C05483=1193.116,-1.564,-43.969,-179.862,5.690,148.965
C05484=1193.121,-1.815,-43.955,-179.864,5.690,148.966
C05485=1193.126,-2.064,-43.941,-179.867,5.690,148.966
C05486=1193.131,-2.313,-43.928,-179.870,5.689,148.967
C05487=1193.136,-2.563,-43.914,-179.872,5.688,148.967
C05488=1193.141,-2.813,-43.900,-179.874,5.688,148.968
C05489=1193.146,-3.062,-43.886,-179.877,5.687,148.969
C05490=1193.151,-3.312,-43.873,-179.880,5.687,148.969
C05491=1193.156,-3.561,-43.859,-179.882,5.686,148.970
C05492=1193.161,-3.811,-43.845,-179.884,5.686,148.971
C05493=1193.166,-4.061,-43.832,-179.887,5.686,148.971
C05494=1193.172,-4.310,-43.818,-179.889,5.685,148.972
C05495=1193.177,-4.560,-43.804,-179.892,5.685,148.973
C05496=1193.182,-4.809,-43.791,-179.895,5.684,148.973
C05497=1193.187,-5.059,-43.777,-179.897,5.683,148.974
C05498=1193.192,-5.309,-43.763,-179.899,5.683,148.974
C05499=1193.197,-5.558,-43.750,-179.902,5.682,148.975
C05500=1193.202,-5.808,-43.736,-179.905,5.682,148.976
C05501=1193.207,-6.057,-43.722,-179.906,5.682,148.976
C05502=1193.212,-6.307,-43.709,-179.909,5.681,148.977
C05503=1193.218,-6.556,-43.695,-179.912,5.681,148.978
C05504=1193.222,-6.806,-43.682,-179.914,5.681,148.978
C05505=1193.227,-7.056,-43.668,-179.917,5.680,148.979
C05506=1193.233,-7.305,-43.655,-179.919,5.679,148.980
C05507=1193.237,-7.555,-43.641,-179.922,5.679,148.980
C05508=1193.243,-7.804,-43.628,-179.924,5.678,148.981
C05509=1193.248,-8.054,-43.614,-179.926,5.679,148.982
C05510=1193.253,-8.303,-43.601,-179.929,5.678,148.982
C05511=1193.258,-8.553,-43.587,-179.931,5.677,148.983
C05512=1193.263,-8.802,-43.574,-179.934,5.677,148.983
C05513=1193.268,-9.052,-43.560,-179.937,5.676,148.984
C05514=1193.273,-9.301,-43.547,-179.939,5.676,148.985
C05515=1193.278,-9.551,-43.533,-179.941,5.675,148.985
C05516=1193.284,-9.801,-43.520,-179.944,5.674,148.986
C05517=1193.289,-10.051,-43.507,-179.946,5.675,148.987
C05518=1193.294,-10.300,-43.493,-179.949,5.674,148.987
C05519=1193.299,-10.550,-43.480,-179.951,5.674,148.988
C05520=1193.304,-10.799,-43.466,-179.954,5.673,148.989
C05521=1193.309,-11.049,-43.453,-179.956,5.673,148.989
C05522=1193.315,-11.298,-43.440,-179.959,5.672,148.990
C05523=1193.319,-11.548,-43.426,-179.962,5.672,148.991
C05524=1193.325,-11.797,-43.413,-179.964,5.672,148.991
C05525=1193.329,-12.048,-43.400,-179.966,5.671,148.992
C05526=1193.335,-12.297,-43.386,-179.968,5.671,148.992
C05527=1193.339,-12.547,-43.373,-179.971,5.670,148.993
C05528=1193.345,-12.796,-43.359,-179.974,5.670,148.994
C05529=1193.349,-13.046,-43.346,-179.976,5.669,148.994
C05530=1193.355,-13.295,-43.333,-179.979,5.668,148.995
C05531=1193.360,-13.545,-43.320,-179.981,5.669,148.996
C05532=1193.365,-13.794,-43.306,-179.983,5.668,148.996
C05533=1193.370,-14.044,-43.293,-179.986,5.668,148.997
C05534=1193.376,-14.294,-43.280,-179.988,5.667,148.998
C05535=1193.380,-14.543,-43.267,-179.991,5.666,148.998
C05536=1193.386,-14.793,-43.253,-179.993,5.666,148.999
C05537=1193.391,-15.042,-43.241,-179.996,5.665,149.000
C05538=1193.395,-15.292,-43.228,-179.998,5.666,149.000
C05539=1193.401,-15.541,-43.214,180.000,5.665,149.001
C05540=1193.405,-15.791,-43.201,179.997,5.664,149.002
C05541=1193.411,-16.041,-43.188,179.994,5.664,149.002
C05542=1193.416,-16.290,-43.175,179.992,5.664,149.003
C05543=1193.421,-16.540,-43.161,179.989,5.663,149.004
C05544=1193.426,-16.789,-43.148,179.987,5.663,149.004
C05545=1193.431,-17.039,-43.135,179.985,5.663,149.005
C05546=1193.437,-17.289,-43.122,179.982,5.662,149.005
C05547=1193.442,-17.538,-43.109,179.979,5.662,149.006
C05548=1193.447,-17.788,-43.096,179.977,5.661,149.007
C05549=1193.452,-18.037,-43.083,179.975,5.660,149.007
C05550=1193.457,-18.287,-43.070,179.973,5.661,149.008
C05551=1193.462,-18.537,-43.056,179.970,5.660,149.009
C05552=1193.468,-18.786,-43.044,179.967,5.660,149.009
C05553=1193.472,-19.036,-43.031,179.965,5.659,149.010
C05554=1193.478,-19.286,-43.018,179.962,5.658,149.011
C05555=1193.483,-19.535,-43.005,179.960,5.658,149.011
C05556=1193.487,-19.785,-42.991,179.958,5.658,149.012
C05557=1193.493,-20.034,-42.978,179.955,5.658,149.013
C05558=1193.498,-20.284,-42.965,179.953,5.657,149.013
C05559=1193.503,-20.534,-42.953,179.950,5.656,149.014
C05560=1193.509,-20.783,-42.939,179.947,5.656,149.014
C05561=1193.513,-21.033,-42.926,179.945,5.656,149.015
C05562=1193.518,-21.282,-42.914,179.943,5.656,149.016
C05563=1193.524,-21.532,-42.901,179.941,5.655,149.016
C05564=1193.529,-21.782,-42.888,179.938,5.655,149.017
C05565=1193.534,-22.031,-42.875,179.935,5.654,149.018
C05566=1193.539,-22.281,-42.862,179.933,5.654,149.018
C05567=1193.544,-22.531,-42.849,179.931,5.654,149.019
C05568=1193.549,-22.780,-42.836,179.928,5.653,149.020
C05569=1193.555,-23.050,-42.822,179.926,5.653,149.020
C05570=1193.561,-23.319,-42.809,179.923,5.652,149.021
C05571=1193.566,-23.590,-42.794,179.920,5.652,149.022
C05572=1193.571,-23.859,-42.780,179.918,5.651,149.022
C05573=1193.576,-24.108,-42.767,179.915,5.651,149.023
C05574=1193.582,-24.358,-42.756,179.912,5.650,149.024
C05575=1193.588,-24.608,-42.742,179.910,5.651,149.024
C05576=1193.592,-24.858,-42.729,179.908,5.650,149.025
C05577=1193.597,-25.107,-42.717,179.905,5.649,149.026
C05578=1193.602,-25.356,-42.704,179.903,5.649,149.026
C05579=1193.608,-25.607,-42.691,179.900,5.648,149.027
C05580=1193.613,-25.856,-42.678,179.898,5.649,149.028
C05581=1193.618,-26.105,-42.665,179.895,5.648,149.028
C05582=1193.623,-26.354,-42.653,179.893,5.647,149.029
C05583=1193.627,-26.604,-42.640,179.891,5.647,149.030
C05584=1193.633,-26.854,-42.627,179.888,5.647,149.030
C05585=1193.638,-27.103,-42.614,179.886,5.647,149.031
C05586=1193.644,-27.353,-42.601,179.883,5.646,149.032
C05587=1193.648,-27.603,-42.589,179.881,5.646,149.032
C05588=1193.654,-27.853,-42.577,179.878,5.645,149.033
C05589=1193.659,-28.102,-42.564,179.876,5.645,149.034
C05590=1193.664,-28.351,-42.551,179.874,5.645,149.034
C05591=1193.669,-28.602,-42.538,179.871,5.644,149.035
C05592=1193.674,-28.851,-42.525,179.869,5.644,149.035
C05593=1193.680,-29.101,-42.513,179.866,5.643,149.036
C05594=1193.685,-29.350,-42.501,179.864,5.644,149.037
C05595=1193.689,-29.600,-42.488,179.861,5.643,149.037
C05596=1193.694,-29.850,-42.475,179.859,5.642,149.038
C05597=1193.699,-30.099,-42.463,179.857,5.642,149.039
C05598=1193.705,-30.349,-42.451,179.854,5.641,149.039
C05599=1193.710,-30.598,-42.438,179.852,5.642,149.040
C05600=1193.715,-30.848,-42.425,179.849,5.641,149.041
C05601=1193.720,-31.098,-42.412,179.847,5.640,149.041
C05602=1193.726,-31.347,-42.399,179.844,5.640,149.042
C05603=1193.731,-31.597,-42.387,179.842,5.640,149.043
C05604=1193.736,-31.846,-42.375,179.840,5.640,149.043
C05605=1193.741,-32.096,-42.362,179.837,5.639,149.044
C05606=1193.746,-32.346,-42.350,179.835,5.639,149.044
C05607=1193.751,-32.596,-42.337,179.832,5.638,149.045
C05608=1193.756,-32.845,-42.325,179.830,5.638,149.046
C05609=1193.761,-33.094,-42.312,179.827,5.638,149.047
C05610=1193.767,-33.344,-42.300,179.825,5.638,149.047
C05611=1193.771,-33.594,-42.287,179.822,5.637,149.048
C05612=1193.776,-33.844,-42.275,179.820,5.637,149.048
C05613=1193.782,-34.093,-42.263,179.818,5.637,149.049
C05614=1193.787,-34.343,-42.250,179.815,5.636,149.050
C05615=1193.792,-34.592,-42.238,179.813,5.635,149.050
C05616=1193.798,-34.842,-42.226,179.811,5.636,149.051
C05617=1193.802,-35.092,-42.213,179.808,5.635,149.052
C05618=1193.807,-35.341,-42.200,179.806,5.635,149.052
C05619=1193.813,-35.591,-42.188,179.803,5.634,149.053
C05620=1193.818,-35.841,-42.176,179.801,5.634,149.054
C05621=1193.823,-36.091,-42.164,179.799,5.634,149.054
C05622=1193.828,-36.340,-42.151,179.796,5.633,149.055
C05623=1193.833,-36.589,-42.139,179.793,5.633,149.056
C05624=1193.839,-36.839,-42.127,179.791,5.633,149.056
C05625=1193.844,-37.088,-42.114,179.789,5.632,149.057
C05626=1193.849,-37.339,-42.102,179.786,5.632,149.058
C05627=1193.854,-37.588,-42.089,179.784,5.632,149.058
C05628=1193.859,-37.838,-42.077,179.782,5.632,149.059
C05629=1193.865,-38.088,-42.065,179.779,5.631,149.060
C05630=1193.870,-38.337,-42.052,179.777,5.631,149.060
C05631=1193.875,-38.587,-42.040,179.774,5.630,149.061
C05632=1193.880,-38.836,-42.028,179.772,5.630,149.062
C05633=1193.886,-39.086,-42.016,179.769,5.630,149.062
C05634=1193.891,-39.335,-42.003,179.767,5.629,149.063
C05635=1193.896,-39.585,-41.991,179.765,5.629,149.063
C05636=1193.901,-39.835,-41.979,179.762,5.629,149.064
C05637=1193.906,-40.084,-41.967,179.760,5.629,149.065
C05638=1193.911,-40.334,-41.954,179.757,5.628,149.065
C05639=1193.916,-40.584,-41.943,179.755,5.627,149.066
C05640=1193.921,-40.834,-41.930,179.753,5.628,149.067
C05641=1193.927,-41.084,-41.918,179.750,5.627,149.067
C05642=1193.932,-41.334,-41.906,179.748,5.627,149.068
C05643=1193.937,-41.583,-41.894,179.745,5.626,149.069
C05644=1193.942,-41.832,-41.882,179.743,5.626,149.069
C05645=1193.947,-42.082,-41.870,179.741,5.626,149.070
C05646=1193.952,-42.332,-41.858,179.738,5.625,149.071
C05647=1193.957,-42.581,-41.845,179.736,5.626,149.071
C05648=1193.963,-42.831,-41.833,179.733,5.625,149.072
C05649=1193.968,-43.081,-41.821,179.731,5.625,149.073
C05650=1193.973,-43.330,-41.809,179.728,5.624,149.073
C05651=1193.978,-43.580,-41.798,179.726,5.624,149.074
C05652=1193.983,-43.829,-41.785,179.724,5.624,149.075
C05653=1193.989,-44.079,-41.773,179.721,5.623,149.075
C05654=1193.994,-44.329,-41.761,179.719,5.623,149.076
C05655=1193.999,-44.578,-41.749,179.717,5.623,149.076
C05656=1194.004,-44.828,-41.737,179.714,5.623,149.077
C05657=1194.009,-45.078,-41.725,179.711,5.622,149.078
C05658=1194.014,-45.327,-41.713,179.710,5.622,149.078
C05659=1194.020,-45.577,-41.701,179.707,5.622,149.079
C05660=1194.025,-45.827,-41.690,179.704,5.621,149.080
C05661=1194.030,-46.076,-41.677,179.702,5.621,149.080
C05662=1194.035,-46.326,-41.665,179.700,5.621,149.081
C05663=1194.041,-46.576,-41.653,179.698,5.620,149.082
C05664=1194.046,-46.825,-41.641,179.695,5.620,149.082
C05665=1194.050,-47.075,-41.629,179.693,5.620,149.083
C05666=1194.056,-47.325,-41.618,179.690,5.620,149.084
C05667=1194.061,-47.575,-41.606,179.688,5.619,149.084
C05668=1194.066,-47.824,-41.594,179.685,5.619,149.085
C05669=1194.071,-48.074,-41.582,179.683,5.619,149.086
C05670=1194.076,-48.324,-41.570,179.681,5.618,149.086
C05671=1194.082,-48.574,-41.558,179.678,5.618,149.087
C05672=1194.086,-48.823,-41.546,179.676,5.618,149.088
C05673=1194.092,-49.092,-41.533,179.674,5.618,149.088
C05674=1194.099,-49.364,-41.521,179.671,5.617,149.089
C05675=1194.104,-49.634,-41.508,179.668,5.617,149.090
C05676=1194.110,-49.904,-41.495,179.666,5.616,149.090
C05677=1194.114,-50.153,-41.484,179.664,5.617,149.091
C05678=1194.120,-50.403,-41.471,179.661,5.616,149.092
C05679=1194.125,-50.652,-41.459,179.658,5.616,149.092
C05680=1194.130,-50.902,-41.448,179.657,5.616,149.093
C05681=1194.135,-51.152,-41.436,179.654,5.615,149.094
C05682=1194.141,-51.402,-41.424,179.651,5.615,149.094
C05683=1194.145,-51.652,-41.413,179.649,5.614,149.095
C05684=1194.151,-51.900,-41.401,179.647,5.615,149.096
C05685=1194.156,-52.150,-41.389,179.644,5.614,149.096
C05686=1194.161,-52.400,-41.377,179.642,5.613,149.097
C05687=1194.167,-52.650,-41.366,179.640,5.614,149.098
C05688=1194.171,-52.899,-41.354,179.637,5.613,149.098
C05689=1194.177,-53.149,-41.342,179.635,5.613,149.099
C05690=1194.182,-53.399,-41.330,179.633,5.613,149.099
C05691=1194.187,-53.649,-41.319,179.630,5.612,149.100
C05692=1194.192,-53.899,-41.307,179.627,5.612,149.101
C05693=1194.198,-54.148,-41.296,179.625,5.612,149.102
C05694=1194.203,-54.397,-41.284,179.623,5.612,149.102
C05695=1194.208,-54.647,-41.272,179.620,5.611,149.103
C05696=1194.213,-54.897,-41.261,179.618,5.611,149.103
C05697=1194.218,-55.146,-41.249,179.616,5.611,149.104
C05698=1194.223,-55.396,-41.237,179.613,5.610,149.105
C05699=1194.228,-55.646,-41.226,179.611,5.610,149.105
C05700=1194.234,-55.895,-41.215,179.609,5.610,149.106
C05701=1194.239,-56.145,-41.203,179.606,5.610,149.107
C05702=1194.244,-56.395,-41.191,179.603,5.609,149.107
C05703=1194.249,-56.644,-41.180,179.602,5.609,149.108
C05704=1194.255,-56.894,-41.168,179.599,5.609,149.109
C05705=1194.259,-57.144,-41.156,179.596,5.608,149.109
C05706=1194.265,-57.394,-41.145,179.594,5.609,149.110
C05707=1194.270,-57.643,-41.134,179.592,5.608,149.111
C05708=1194.275,-57.893,-41.122,179.590,5.607,149.111
C05709=1194.280,-58.142,-41.110,179.587,5.608,149.112
C05710=1194.286,-58.392,-41.099,179.585,5.607,149.113
C05711=1194.290,-58.642,-41.087,179.583,5.607,149.113
C05712=1194.296,-58.891,-41.076,179.581,5.607,149.114
C05713=1194.301,-59.142,-41.065,179.578,5.606,149.115
C05714=1194.307,-59.391,-41.053,179.575,5.606,149.115
C05715=1194.311,-59.641,-41.042,179.573,5.606,149.116
C05716=1194.316,-59.891,-41.031,179.571,5.606,149.116
C05717=1194.322,-60.140,-41.019,179.568,5.605,149.117
C05718=1194.327,-60.390,-41.008,179.566,5.606,149.118
C05719=1194.332,-60.639,-40.996,179.564,5.605,149.119
C05720=1194.337,-60.889,-40.985,179.561,5.604,149.119
C05721=1194.342,-61.139,-40.973,179.559,5.605,149.120
C05722=1194.348,-61.388,-40.962,179.557,5.604,149.120
C05723=1194.353,-61.639,-40.951,179.554,5.604,149.121
C05724=1194.358,-61.888,-40.939,179.552,5.604,149.122
C05725=1194.363,-62.138,-40.928,179.550,5.603,149.122
C05726=1194.369,-62.387,-40.917,179.548,5.604,149.123
C05727=1194.373,-62.637,-40.905,179.545,5.603,149.124
C05728=1194.379,-62.887,-40.893,179.543,5.602,149.124
C05729=1194.384,-63.137,-40.883,179.541,5.603,149.125
C05730=1194.390,-63.386,-40.871,179.538,5.602,149.126
C05731=1194.395,-63.636,-40.860,179.535,5.602,149.126
C05732=1194.399,-63.885,-40.849,179.534,5.602,149.127
C05733=1194.405,-64.135,-40.837,179.531,5.601,149.128
C05734=1194.410,-64.385,-40.827,179.528,5.601,149.128
C05735=1194.416,-64.635,-40.815,179.526,5.601,149.129
C05736=1194.420,-64.884,-40.803,179.524,5.601,149.129
C05737=1194.426,-65.133,-40.793,179.521,5.600,149.130
C05738=1194.431,-65.384,-40.781,179.519,5.601,149.131
C05739=1194.436,-65.633,-40.770,179.517,5.600,149.132
C05740=1194.441,-65.883,-40.759,179.514,5.600,149.132
C05741=1194.447,-66.132,-40.747,179.512,5.600,149.133
C05742=1194.452,-66.383,-40.737,179.510,5.599,149.133
C05743=1194.457,-66.632,-40.725,179.508,5.600,149.134
C05744=1194.463,-66.881,-40.714,179.505,5.599,149.135
C05745=1194.468,-67.132,-40.703,179.503,5.598,149.135
C05746=1194.472,-67.381,-40.692,179.501,5.599,149.136
C05747=1194.478,-67.631,-40.681,179.498,5.598,149.137
C05748=1194.483,-67.881,-40.670,179.495,5.598,149.137
C05749=1194.488,-68.130,-40.659,179.494,5.598,149.138
C05750=1194.494,-68.380,-40.647,179.491,5.597,149.139
C05751=1194.499,-68.630,-40.637,179.488,5.597,149.139
C05752=1194.504,-68.880,-40.625,179.486,5.597,149.140
C05753=1194.509,-69.128,-40.614,179.484,5.597,149.141
C05754=1194.515,-69.379,-40.603,179.482,5.597,149.141
C05755=1194.519,-69.629,-40.592,179.479,5.596,149.142
C05756=1194.525,-69.878,-40.581,179.477,5.596,149.143
C05757=1194.531,-70.128,-40.570,179.475,5.596,149.143
C05758=1194.535,-70.378,-40.559,179.473,5.596,149.144
C05759=1194.541,-70.627,-40.548,179.470,5.595,149.145
C05760=1194.545,-70.877,-40.537,179.468,5.596,149.145
C05761=1194.551,-71.127,-40.525,179.466,5.595,149.146
C05762=1194.557,-71.376,-40.515,179.463,5.595,149.146
C05763=1194.561,-71.626,-40.504,179.461,5.595,149.147
C05764=1194.567,-71.876,-40.493,179.459,5.594,149.148
C05765=1194.572,-72.125,-40.482,179.457,5.594,149.148
C05766=1194.577,-72.376,-40.471,179.454,5.594,149.149
C05767=1194.583,-72.625,-40.460,179.451,5.593,149.150
C05768=1194.588,-72.875,-40.449,179.450,5.593,149.150
C05769=1194.593,-73.124,-40.439,179.447,5.593,149.151
C05770=1194.599,-73.374,-40.427,179.445,5.593,149.152
C05771=1194.603,-73.624,-40.416,179.442,5.593,149.152
C05772=1194.609,-73.874,-40.406,179.440,5.592,149.153
C05773=1194.614,-74.123,-40.395,179.438,5.592,149.154
C05774=1194.619,-74.373,-40.384,179.435,5.592,149.154
C05775=1194.625,-74.623,-40.372,179.433,5.592,149.155
C05776=1194.630,-74.873,-40.362,179.431,5.592,149.155
C05777=1194.636,-75.143,-40.350,179.428,5.591,149.156
C05778=1194.641,-75.414,-40.338,179.426,5.591,149.157
C05779=1194.646,-75.685,-40.326,179.424,5.591,149.158
C05780=1194.653,-75.956,-40.315,179.421,5.591,149.158
C05781=1194.657,-76.205,-40.304,179.418,5.590,149.159
C05782=1194.663,-76.455,-40.293,179.416,5.591,149.160
C05783=1194.668,-76.705,-40.282,179.414,5.590,149.160
C05784=1194.673,-76.954,-40.272,179.412,5.590,149.161
C05785=1194.678,-77.204,-40.261,179.409,5.590,149.162
C05786=1194.684,-77.453,-40.250,179.407,5.589,149.162
C05787=1194.689,-77.704,-40.239,179.405,5.589,149.163
C05788=1194.694,-77.953,-40.228,179.402,5.589,149.163
C05789=1194.700,-78.203,-40.218,179.400,5.589,149.164
C05790=1194.705,-78.453,-40.207,179.397,5.589,149.165
C05791=1194.710,-78.702,-40.196,179.395,5.588,149.165
C05792=1194.715,-78.952,-40.186,179.393,5.589,149.166
C05793=1194.720,-79.201,-40.175,179.391,5.588,149.167
C05794=1194.725,-79.452,-40.164,179.389,5.588,149.167
C05795=1194.731,-79.701,-40.154,179.386,5.588,149.168
C05796=1194.736,-79.951,-40.143,179.384,5.587,149.169
C05797=1194.741,-80.200,-40.133,179.382,5.588,149.169
C05798=1194.746,-80.450,-40.122,179.379,5.587,149.170
C05799=1194.752,-80.700,-40.110,179.377,5.587,149.171
C05800=1194.757,-80.950,-40.100,179.375,5.587,149.171
C05801=1194.763,-81.200,-40.090,179.372,5.586,149.172
C05802=1194.768,-81.450,-40.079,179.370,5.586,149.172
C05803=1194.773,-81.699,-40.068,179.368,5.586,149.173
C05804=1194.778,-81.949,-40.058,179.366,5.586,149.174
C05805=1194.784,-82.198,-40.047,179.363,5.586,149.174
C05806=1194.788,-82.448,-40.036,179.361,5.585,149.175
C05807=1194.794,-82.698,-40.026,179.359,5.585,149.176
C05808=1194.799,-82.948,-40.015,179.356,5.585,149.176
C05809=1194.805,-83.197,-40.005,179.354,5.585,149.177
C05810=1194.809,-83.447,-39.994,179.352,5.585,149.178
C05811=1194.815,-83.697,-39.984,179.350,5.585,149.178
C05812=1194.820,-83.947,-39.973,179.347,5.584,149.179
C05813=1194.825,-84.196,-39.963,179.345,5.584,149.180
C05814=1194.831,-84.446,-39.953,179.343,5.584,149.180
C05815=1194.836,-84.696,-39.941,179.340,5.583,149.181
C05816=1194.841,-84.945,-39.931,179.338,5.584,149.181
C05817=1194.846,-85.195,-39.920,179.336,5.583,149.182
C05818=1194.852,-85.445,-39.910,179.334,5.584,149.183
C05819=1194.856,-85.695,-39.900,179.331,5.583,149.183
C05820=1194.861,-85.944,-39.889,179.329,5.583,149.184
C05821=1194.866,-86.194,-39.879,179.327,5.583,149.185
C05822=1194.872,-86.444,-39.869,179.324,5.582,149.185
C05823=1194.878,-86.693,-39.858,179.322,5.582,149.186
C05824=1194.883,-86.943,-39.848,179.320,5.582,149.187
C05825=1194.888,-87.193,-39.838,179.318,5.582,149.187
C05826=1194.893,-87.442,-39.826,179.315,5.582,149.188
C05827=1194.899,-87.692,-39.816,179.313,5.581,149.189
C05828=1194.904,-87.942,-39.806,179.311,5.582,149.189
C05829=1194.909,-88.192,-39.795,179.309,5.581,149.190
C05830=1194.915,-88.441,-39.785,179.306,5.581,149.191
C05831=1194.919,-88.691,-39.775,179.304,5.581,149.191
C05832=1194.925,-88.941,-39.765,179.302,5.581,149.192
C05833=1194.930,-89.190,-39.755,179.299,5.580,149.192
C05834=1194.935,-89.441,-39.744,179.297,5.580,149.193
C05835=1194.941,-89.690,-39.734,179.295,5.580,149.194
C05836=1194.946,-89.940,-39.723,179.293,5.580,149.194
C05837=1194.951,-90.190,-39.713,179.290,5.580,149.195
C05838=1194.957,-90.439,-39.702,179.288,5.579,149.196
C05839=1194.961,-90.689,-39.692,179.286,5.579,149.196
C05840=1194.967,-90.938,-39.682,179.284,5.579,149.197
C05841=1194.972,-91.188,-39.672,179.281,5.579,149.198
C05842=1194.977,-91.438,-39.661,179.279,5.579,149.198
C05843=1194.983,-91.688,-39.651,179.277,5.578,149.199
C05844=1194.988,-91.938,-39.640,179.274,5.579,149.200
C05845=1194.993,-92.187,-39.631,179.272,5.578,149.200
C05846=1194.998,-92.437,-39.621,179.270,5.578,149.201
C05847=1195.003,-92.687,-39.610,179.268,5.578,149.201
C05848=1195.009,-92.936,-39.600,179.265,5.578,149.202
C05849=1195.014,-93.186,-39.590,179.263,5.577,149.203
C05850=1195.019,-93.436,-39.580,179.261,5.578,149.203
C05851=1195.024,-93.686,-39.569,179.259,5.577,149.204
C05852=1195.030,-93.936,-39.560,179.256,5.577,149.205
C05853=1195.035,-94.186,-39.549,179.254,5.577,149.205
C05854=1195.041,-94.435,-39.539,179.252,5.577,149.206
C05855=1195.046,-94.685,-39.530,179.250,5.577,149.206
C05856=1195.051,-94.935,-39.519,179.247,5.576,149.207
C05857=1195.056,-95.184,-39.509,179.245,5.577,149.208
C05858=1195.062,-95.434,-39.499,179.243,5.576,149.208
C05859=1195.067,-95.683,-39.489,179.241,5.576,149.209
C05860=1195.072,-95.934,-39.478,179.238,5.576,149.210
C05861=1195.077,-96.183,-39.468,179.236,5.575,149.210
C05862=1195.083,-96.433,-39.458,179.234,5.575,149.211
C05863=1195.087,-96.683,-39.449,179.231,5.575,149.212
C05864=1195.093,-96.933,-39.439,179.230,5.575,149.212
C05865=1195.099,-97.182,-39.428,179.227,5.575,149.213
C05866=1195.104,-97.432,-39.418,179.225,5.575,149.214
C05867=1195.108,-97.682,-39.408,179.223,5.574,149.214
C05868=1195.114,-97.931,-39.398,179.221,5.574,149.215
C05869=1195.120,-98.181,-39.388,179.218,5.574,149.216
C05870=1195.125,-98.432,-39.378,179.216,5.574,149.216
C05871=1195.130,-98.681,-39.368,179.214,5.574,149.217
C05872=1195.135,-98.930,-39.358,179.212,5.574,149.217
C05873=1195.141,-99.180,-39.348,179.209,5.573,149.218
C05874=1195.145,-99.430,-39.338,179.207,5.573,149.219
C05875=1195.151,-99.680,-39.328,179.205,5.573,149.219
C05876=1195.157,-99.930,-39.318,179.202,5.572,149.220
C05877=1195.162,-100.179,-39.309,179.200,5.573,149.221
C05878=1195.167,-100.429,-39.298,179.198,5.572,149.221
C05879=1195.172,-100.679,-39.288,179.196,5.572,149.222
C05880=1195.177,-100.928,-39.279,179.193,5.572,149.222
C05881=1195.183,-101.200,-39.267,179.191,5.572,149.223
C05882=1195.189,-101.471,-39.256,179.189,5.572,149.224
C05883=1195.195,-101.743,-39.247,179.186,5.572,149.225
C05884=1195.201,-102.014,-39.235,179.184,5.572,149.225
C05885=1195.206,-102.264,-39.226,179.182,5.571,149.226
C05886=1195.211,-102.514,-39.216,179.180,5.572,149.227
C05887=1195.216,-102.764,-39.206,179.177,5.571,149.227
C05888=1195.221,-103.013,-39.196,179.175,5.571,149.228
C05889=1195.227,-103.263,-39.186,179.173,5.571,149.228
C05890=1195.232,-103.512,-39.177,179.171,5.570,149.229
C05891=1195.238,-103.762,-39.166,179.168,5.570,149.230
C05892=1195.242,-104.013,-39.157,179.166,5.570,149.230
C05893=1195.248,-104.262,-39.147,179.164,5.570,149.231
C05894=1195.253,-104.512,-39.137,179.161,5.570,149.232
C05895=1195.258,-104.762,-39.128,179.159,5.570,149.232
C05896=1195.264,-105.011,-39.118,179.157,5.569,149.233
C05897=1195.268,-105.261,-39.108,179.155,5.570,149.233
C05898=1195.274,-105.511,-39.098,179.152,5.569,149.234
C05899=1195.279,-105.760,-39.088,179.151,5.569,149.235
C05900=1195.285,-106.010,-39.078,179.148,5.569,149.235
C05901=1195.291,-106.260,-39.069,179.146,5.569,149.236
C05902=1195.295,-106.509,-39.059,179.144,5.568,149.237
C05903=1195.301,-106.760,-39.049,179.142,5.569,149.237
C05904=1195.306,-107.009,-39.040,179.140,5.568,149.238
C05905=1195.311,-107.259,-39.029,179.138,5.568,149.238
C05906=1195.316,-107.509,-39.021,179.135,5.568,149.239
C05907=1195.322,-107.758,-39.010,179.133,5.568,149.240
C05908=1195.327,-108.008,-39.001,179.131,5.568,149.240
C05909=1195.332,-108.258,-38.991,179.128,5.568,149.241
C05910=1195.337,-108.508,-38.982,179.126,5.567,149.242
C05911=1195.343,-108.758,-38.972,179.124,5.568,149.242
C05912=1195.348,-109.007,-38.962,179.122,5.567,149.243
C05913=1195.354,-109.257,-38.953,179.120,5.567,149.243
C05914=1195.359,-109.506,-38.943,179.117,5.567,149.244
C05915=1195.364,-109.757,-38.934,179.116,5.567,149.245
C05916=1195.369,-110.006,-38.924,179.113,5.566,149.245
C05917=1195.375,-110.257,-38.914,179.111,5.567,149.246
C05918=1195.379,-110.506,-38.905,179.109,5.566,149.247
C05919=1195.385,-110.756,-38.895,179.107,5.566,149.247
C05920=1195.390,-111.005,-38.885,179.104,5.566,149.248
C05921=1195.396,-111.256,-38.876,179.102,5.566,149.249
C05922=1195.401,-111.505,-38.866,179.100,5.566,149.249
C05923=1195.406,-111.755,-38.857,179.098,5.566,149.250
C05924=1195.412,-112.004,-38.847,179.095,5.565,149.250
C05925=1195.417,-112.254,-38.838,179.093,5.566,149.251
C05926=1195.423,-112.504,-38.828,179.091,5.565,149.252
C05927=1195.428,-112.753,-38.819,179.089,5.565,149.252
C05928=1195.433,-113.004,-38.809,179.087,5.565,149.253
C05929=1195.438,-113.254,-38.800,179.085,5.565,149.254
C05930=1195.443,-113.503,-38.791,179.082,5.565,149.254
C05931=1195.449,-113.753,-38.781,179.080,5.565,149.255
C05932=1195.454,-114.003,-38.772,179.078,5.564,149.255
C05933=1195.459,-114.252,-38.761,179.076,5.564,149.256
C05934=1195.465,-114.502,-38.753,179.074,5.564,149.257
C05935=1195.470,-114.752,-38.744,179.071,5.564,149.257
C05936=1195.475,-115.002,-38.733,179.069,5.563,149.258
C05937=1195.480,-115.251,-38.725,179.067,5.564,149.259
C05938=1195.486,-115.502,-38.715,179.065,5.563,149.259
C05939=1195.491,-115.751,-38.705,179.063,5.563,149.260
C05940=1195.496,-116.001,-38.697,179.060,5.563,149.260
C05941=1195.502,-116.250,-38.686,179.059,5.563,149.261
C05942=1195.507,-116.500,-38.677,179.056,5.563,149.262
C05943=1195.512,-116.750,-38.669,179.054,5.563,149.262
C05944=1195.518,-116.999,-38.658,179.052,5.562,149.263
C05945=1195.523,-117.249,-38.649,179.050,5.563,149.264
C05946=1195.528,-117.499,-38.641,179.047,5.562,149.264
C05947=1195.534,-117.749,-38.630,179.045,5.562,149.265
C05948=1195.539,-117.999,-38.621,179.043,5.561,149.265
C05949=1195.544,-118.248,-38.613,179.041,5.562,149.266
C05950=1195.550,-118.499,-38.603,179.038,5.561,149.267
C05951=1195.555,-118.748,-38.593,179.037,5.561,149.267
C05952=1195.560,-118.998,-38.585,179.034,5.561,149.268
C05953=1195.566,-119.248,-38.575,179.032,5.561,149.268
C05954=1195.571,-119.497,-38.565,179.030,5.561,149.269
C05955=1195.576,-119.747,-38.557,179.028,5.561,149.270
C05956=1195.582,-119.997,-38.547,179.025,5.560,149.270
C05957=1195.587,-120.247,-38.538,179.023,5.561,149.271
C05958=1195.592,-120.496,-38.529,179.021,5.560,149.272
C05959=1195.597,-120.746,-38.520,179.019,5.560,149.272
C05960=1195.603,-120.996,-38.510,179.017,5.560,149.273
C05961=1195.608,-121.246,-38.501,179.015,5.560,149.273
C05962=1195.613,-121.495,-38.492,179.013,5.560,149.274
C05963=1195.618,-121.745,-38.483,179.011,5.560,149.275
C05964=1195.624,-121.995,-38.473,179.008,5.560,149.275
C05965=1195.629,-122.245,-38.464,179.006,5.559,149.276
C05966=1195.635,-122.495,-38.455,179.004,5.560,149.277
C05967=1195.639,-122.744,-38.446,179.002,5.559,149.277
C05968=1195.645,-122.994,-38.436,179.000,5.559,149.278
C05969=1195.650,-123.244,-38.427,178.997,5.559,149.278
C05970=1195.656,-123.494,-38.419,178.996,5.559,149.279
C05971=1195.661,-123.744,-38.410,178.993,5.558,149.280
C05972=1195.667,-123.994,-38.400,178.991,5.558,149.280
C05973=1195.672,-124.243,-38.391,178.989,5.558,149.281
C05974=1195.677,-124.493,-38.382,178.987,5.558,149.281
C05975=1195.682,-124.743,-38.373,178.984,5.558,149.282
C05976=1195.687,-124.993,-38.364,178.983,5.558,149.283
C05977=1195.694,-125.242,-38.355,178.980,5.557,149.283
C05978=1195.699,-125.492,-38.346,178.978,5.558,149.284
C05979=1195.704,-125.742,-38.337,178.976,5.557,149.285
C05980=1195.709,-125.992,-38.328,178.974,5.557,149.285
C05981=1195.714,-126.241,-38.318,178.972,5.557,149.286
C05982=1195.719,-126.491,-38.310,178.969,5.557,149.286
C05983=1195.725,-126.741,-38.300,178.968,5.557,149.287
C05984=1195.730,-126.991,-38.291,178.965,5.557,149.288
C05985=1195.309,-127.002,-38.330,178.961,5.560,149.289
C05986=1195.303,-126.752,-38.339,178.963,5.561,149.289
C05987=1195.298,-126.502,-38.348,178.966,5.560,149.288
C05988=1195.293,-126.252,-38.357,178.968,5.561,149.288
C05989=1195.287,-126.002,-38.366,178.970,5.561,149.287
C05990=1195.283,-125.753,-38.376,178.972,5.561,149.286
C05991=1195.277,-125.503,-38.385,178.974,5.561,149.286
C05992=1195.272,-125.253,-38.394,178.977,5.561,149.285
C05993=1195.266,-125.004,-38.403,178.978,5.561,149.285
C05994=1195.261,-124.754,-38.412,178.980,5.561,149.284
C05995=1195.255,-124.504,-38.420,178.983,5.562,149.283
C05996=1195.250,-124.254,-38.429,178.985,5.561,149.283
C05997=1195.244,-124.004,-38.439,178.987,5.562,149.282
C05998=1195.239,-123.755,-38.448,178.989,5.562,149.282
C05999=1195.234,-123.505,-38.457,178.992,5.562,149.281
C06000=1195.229,-123.255,-38.466,178.993,5.562,149.280
C06001=1195.224,-123.005,-38.475,178.996,5.562,149.280
C06002=1195.218,-122.755,-38.485,178.998,5.562,149.279
C06003=1195.213,-122.505,-38.494,179.000,5.563,149.278
C06004=1195.208,-122.256,-38.503,179.002,5.563,149.278
C06005=1195.203,-122.006,-38.512,179.005,5.563,149.277
C06006=1195.197,-121.756,-38.522,179.007,5.563,149.277
C06007=1195.192,-121.506,-38.530,179.009,5.564,149.276
C06008=1195.187,-121.256,-38.539,179.011,5.563,149.275
C06009=1195.182,-121.007,-38.549,179.013,5.564,149.275
C06010=1195.176,-120.757,-38.558,179.015,5.564,149.274
C06011=1195.171,-120.507,-38.567,179.017,5.564,149.274
C06012=1195.166,-120.257,-38.576,179.019,5.564,149.273
C06013=1195.161,-120.008,-38.586,179.022,5.564,149.272
C06014=1195.155,-119.758,-38.595,179.024,5.564,149.272
C06015=1195.150,-119.508,-38.604,179.026,5.564,149.271
C06016=1195.144,-119.258,-38.613,179.028,5.565,149.271
C06017=1195.139,-119.009,-38.623,179.030,5.564,149.270
C06018=1195.134,-118.759,-38.632,179.032,5.565,149.269
C06019=1195.129,-118.509,-38.641,179.034,5.565,149.269
C06020=1195.123,-118.259,-38.651,179.037,5.565,149.268
C06021=1195.118,-118.009,-38.660,179.039,5.565,149.267
C06022=1195.113,-117.760,-38.669,179.041,5.565,149.267
C06023=1195.108,-117.510,-38.679,179.043,5.565,149.266
C06024=1195.102,-117.260,-38.688,179.046,5.566,149.265
C06025=1195.097,-117.010,-38.697,179.048,5.565,149.265
C06026=1195.091,-116.760,-38.707,179.050,5.566,149.264
C06027=1195.086,-116.511,-38.716,179.052,5.566,149.264
C06028=1195.081,-116.261,-38.725,179.054,5.567,149.263
C06029=1195.075,-116.012,-38.735,179.056,5.566,149.262
C06030=1195.070,-115.762,-38.744,179.059,5.567,149.262
C06031=1195.065,-115.512,-38.753,179.061,5.567,149.261
C06032=1195.059,-115.262,-38.763,179.063,5.567,149.260
C06033=1195.054,-115.013,-38.772,179.065,5.567,149.260
C06034=1195.049,-114.763,-38.781,179.068,5.567,149.259
C06035=1195.043,-114.513,-38.791,179.070,5.567,149.259
C06036=1195.038,-114.263,-38.800,179.072,5.568,149.258
C06037=1195.033,-114.014,-38.810,179.074,5.567,149.257
C06038=1195.027,-113.764,-38.819,179.076,5.568,149.257
C06039=1195.022,-113.514,-38.828,179.078,5.568,149.256
C06040=1195.017,-113.264,-38.838,179.081,5.568,149.255
C06041=1195.011,-113.015,-38.847,179.082,5.568,149.255
C06042=1195.006,-112.765,-38.858,179.085,5.568,149.254
C06043=1195.001,-112.515,-38.866,179.087,5.568,149.254
C06044=1194.996,-112.265,-38.877,179.089,5.569,149.253
C06045=1194.990,-112.015,-38.886,179.091,5.568,149.252
C06046=1194.985,-111.765,-38.895,179.094,5.569,149.252
C06047=1194.980,-111.516,-38.905,179.096,5.569,149.251
C06048=1194.975,-111.266,-38.914,179.098,5.570,149.251
C06049=1194.969,-111.016,-38.924,179.100,5.569,149.250
C06050=1194.964,-110.766,-38.933,179.103,5.570,149.249
C06051=1194.958,-110.517,-38.943,179.104,5.570,149.249
C06052=1194.953,-110.267,-38.952,179.107,5.570,149.248
C06053=1194.947,-110.018,-38.962,179.109,5.570,149.247
C06054=1194.942,-109.768,-38.971,179.111,5.570,149.247
C06055=1194.937,-109.517,-38.982,179.113,5.570,149.246
C06056=1194.932,-109.268,-38.991,179.116,5.571,149.246
C06057=1194.926,-109.018,-39.001,179.118,5.570,149.245
C06058=1194.922,-108.769,-39.011,179.120,5.571,149.244
C06059=1194.916,-108.519,-39.020,179.122,5.571,149.244
C06060=1194.911,-108.269,-39.030,179.125,5.571,149.243
C06061=1194.905,-108.019,-39.039,179.126,5.571,149.242
C06062=1194.901,-107.769,-39.049,179.129,5.572,149.242
C06063=1194.895,-107.519,-39.059,179.131,5.571,149.241
C06064=1194.890,-107.270,-39.068,179.133,5.572,149.241
C06065=1194.884,-107.020,-39.078,179.135,5.572,149.240
C06066=1194.879,-106.771,-39.087,179.138,5.572,149.239
C06067=1194.874,-106.521,-39.098,179.139,5.572,149.239
C06068=1194.868,-106.271,-39.106,179.142,5.572,149.238
C06069=1194.863,-106.021,-39.117,179.144,5.572,149.237
C06070=1194.859,-105.772,-39.127,179.146,5.573,149.237
C06071=1194.853,-105.522,-39.136,179.149,5.572,149.236
C06072=1194.848,-105.272,-39.146,179.151,5.573,149.236
C06073=1194.842,-105.022,-39.155,179.153,5.573,149.235
C06074=1194.836,-104.773,-39.165,179.155,5.573,149.234
C06075=1194.832,-104.523,-39.175,179.158,5.574,149.234
C06076=1194.826,-104.272,-39.185,179.160,5.574,149.233
C06077=1194.821,-104.023,-39.195,179.162,5.574,149.232
C06078=1194.816,-103.774,-39.205,179.164,5.574,149.232
C06079=1194.810,-103.524,-39.214,179.167,5.574,149.231
C06080=1194.805,-103.274,-39.224,179.169,5.574,149.230
C06081=1194.800,-103.024,-39.234,179.171,5.575,149.230
C06082=1194.795,-102.775,-39.244,179.173,5.574,149.229
C06083=1194.789,-102.525,-39.254,179.176,5.575,149.228
C06084=1194.784,-102.275,-39.263,179.177,5.575,149.228
C06085=1194.779,-102.025,-39.274,179.180,5.575,149.227
C06086=1194.773,-101.754,-39.284,179.182,5.575,149.226
C06087=1194.767,-101.482,-39.295,179.185,5.575,149.226
C06088=1194.762,-101.210,-39.305,179.187,5.576,149.225
C06089=1194.757,-100.939,-39.316,179.189,5.576,149.225
C06090=1194.751,-100.690,-39.326,179.192,5.576,149.224
C06091=1194.745,-100.440,-39.337,179.194,5.576,149.223
C06092=1194.740,-100.190,-39.346,179.196,5.576,149.223
C06093=1194.735,-99.940,-39.356,179.199,5.577,149.222
C06094=1194.730,-99.690,-39.366,179.201,5.576,149.221
C06095=1194.725,-99.441,-39.376,179.203,5.577,149.221
C06096=1194.719,-99.191,-39.385,179.205,5.577,149.220
C06097=1194.714,-98.941,-39.396,179.208,5.577,149.219
C06098=1194.709,-98.692,-39.406,179.209,5.577,149.219
C06099=1194.703,-98.442,-39.416,179.212,5.578,149.218
C06100=1194.698,-98.192,-39.426,179.214,5.577,149.217
C06101=1194.693,-97.942,-39.437,179.216,5.578,149.217
C06102=1194.688,-97.692,-39.446,179.218,5.578,149.216
C06103=1194.682,-97.443,-39.456,179.221,5.578,149.215
C06104=1194.676,-97.193,-39.466,179.223,5.578,149.215
C06105=1194.672,-96.943,-39.476,179.225,5.578,149.214
C06106=1194.667,-96.694,-39.486,179.228,5.579,149.214
C06107=1194.661,-96.444,-39.496,179.230,5.579,149.213
C06108=1194.656,-96.193,-39.506,179.232,5.579,149.212
C06109=1194.651,-95.944,-39.516,179.234,5.579,149.212
C06110=1194.645,-95.695,-39.526,179.237,5.580,149.211
C06111=1194.640,-95.445,-39.536,179.239,5.579,149.210
C06112=1194.635,-95.195,-39.547,179.241,5.580,149.210
C06113=1194.630,-94.946,-39.556,179.243,5.580,149.209
C06114=1194.624,-94.696,-39.567,179.246,5.580,149.209
C06115=1194.619,-94.446,-39.577,179.248,5.580,149.208
C06116=1194.614,-94.196,-39.587,179.250,5.581,149.207
C06117=1194.608,-93.947,-39.598,179.252,5.581,149.207
C06118=1194.604,-93.697,-39.608,179.255,5.581,149.206
C06119=1194.598,-93.447,-39.618,179.257,5.581,149.205
C06120=1194.593,-93.198,-39.628,179.259,5.581,149.205
C06121=1194.588,-92.947,-39.639,179.262,5.581,149.204
C06122=1194.582,-92.697,-39.648,179.263,5.581,149.204
C06123=1194.577,-92.448,-39.658,179.266,5.582,149.203
C06124=1194.572,-92.198,-39.668,179.268,5.581,149.202
C06125=1194.566,-91.948,-39.679,179.270,5.582,149.202
C06126=1194.561,-91.699,-39.689,179.273,5.583,149.201
C06127=1194.556,-91.448,-39.699,179.275,5.582,149.200
C06128=1194.551,-91.199,-39.709,179.278,5.583,149.200
C06129=1194.545,-90.950,-39.719,179.279,5.583,149.199
C06130=1194.540,-90.700,-39.730,179.282,5.583,149.198
C06131=1194.535,-90.451,-39.741,179.284,5.583,149.198
C06132=1194.530,-90.200,-39.751,179.286,5.583,149.197
C06133=1194.524,-89.951,-39.761,179.288,5.583,149.196
C06134=1194.519,-89.701,-39.772,179.291,5.583,149.196
C06135=1194.514,-89.451,-39.782,179.293,5.584,149.195
C06136=1194.509,-89.202,-39.792,179.295,5.584,149.195
C06137=1194.503,-88.952,-39.802,179.298,5.584,149.194
C06138=1194.498,-88.702,-39.813,179.299,5.584,149.193
C06139=1194.493,-88.452,-39.823,179.302,5.585,149.193
C06140=1194.488,-88.202,-39.833,179.304,5.584,149.192
C06141=1194.482,-87.953,-39.844,179.307,5.585,149.191
C06142=1194.476,-87.703,-39.854,179.309,5.586,149.191
C06143=1194.471,-87.453,-39.864,179.311,5.585,149.190
C06144=1194.467,-87.204,-39.875,179.314,5.586,149.189
C06145=1194.462,-86.954,-39.885,179.315,5.586,149.189
C06146=1194.456,-86.704,-39.895,179.318,5.586,149.188
C06147=1194.451,-86.454,-39.906,179.320,5.586,149.187
C06148=1194.446,-86.205,-39.916,179.322,5.586,149.187
C06149=1194.440,-85.955,-39.926,179.325,5.587,149.186
C06150=1194.435,-85.705,-39.938,179.327,5.586,149.185
C06151=1194.430,-85.456,-39.948,179.330,5.587,149.185
C06152=1194.425,-85.206,-39.959,179.331,5.587,149.184
C06153=1194.419,-84.956,-39.969,179.334,5.587,149.184
C06154=1194.414,-84.706,-39.979,179.336,5.587,149.183
C06155=1194.409,-84.456,-39.990,179.338,5.588,149.182
C06156=1194.404,-84.207,-40.001,179.341,5.588,149.182
C06157=1194.398,-83.957,-40.011,179.343,5.588,149.181
C06158=1194.393,-83.708,-40.021,179.346,5.588,149.180
C06159=1194.388,-83.457,-40.032,179.347,5.588,149.180
C06160=1194.382,-83.208,-40.043,179.350,5.589,149.179
C06161=1194.377,-82.958,-40.053,179.353,5.589,149.178
C06162=1194.372,-82.709,-40.064,179.354,5.589,149.178
C06163=1194.367,-82.458,-40.074,179.357,5.589,149.177
C06164=1194.361,-82.210,-40.085,179.359,5.589,149.176
C06165=1194.356,-81.959,-40.096,179.361,5.590,149.176
C06166=1194.351,-81.710,-40.106,179.363,5.589,149.175
C06167=1194.346,-81.459,-40.116,179.366,5.590,149.175
C06168=1194.341,-81.211,-40.127,179.369,5.590,149.174
C06169=1194.336,-80.960,-40.138,179.370,5.590,149.173
C06170=1194.330,-80.711,-40.148,179.373,5.591,149.173
C06171=1194.325,-80.461,-40.159,179.375,5.590,149.172
C06172=1194.320,-80.212,-40.170,179.378,5.591,149.171
C06173=1194.315,-79.961,-40.180,179.380,5.592,149.171
C06174=1194.309,-79.712,-40.191,179.382,5.591,149.170
C06175=1194.304,-79.462,-40.202,179.385,5.592,149.169
C06176=1194.299,-79.213,-40.212,179.386,5.592,149.169
C06177=1194.294,-78.963,-40.223,179.389,5.592,149.168
C06178=1194.289,-78.713,-40.233,179.391,5.592,149.167
C06179=1194.284,-78.463,-40.244,179.394,5.592,149.167
C06180=1194.278,-78.214,-40.255,179.396,5.593,149.166
C06181=1194.273,-77.964,-40.266,179.398,5.593,149.166
C06182=1194.267,-77.714,-40.276,179.400,5.593,149.165
C06183=1194.262,-77.465,-40.288,179.403,5.594,149.164
C06184=1194.257,-77.214,-40.298,179.405,5.593,149.164
C06185=1194.252,-76.965,-40.309,179.407,5.594,149.163
C06186=1194.247,-76.715,-40.320,179.410,5.593,149.162
C06187=1194.241,-76.466,-40.330,179.412,5.594,149.162
C06188=1194.236,-76.216,-40.342,179.414,5.595,149.161
C06189=1194.230,-75.966,-40.352,179.416,5.594,149.160
C06190=1194.225,-75.695,-40.364,179.419,5.595,149.160
C06191=1194.220,-75.424,-40.376,179.422,5.595,149.159
C06192=1194.213,-75.154,-40.387,179.424,5.595,149.158
C06193=1194.208,-74.883,-40.399,179.427,5.595,149.157
C06194=1194.202,-74.634,-40.410,179.429,5.596,149.157
C06195=1194.197,-74.383,-40.421,179.431,5.596,149.156
C06196=1194.193,-74.134,-40.432,179.434,5.596,149.156
C06197=1194.187,-73.884,-40.442,179.436,5.596,149.155
C06198=1194.182,-73.635,-40.454,179.438,5.596,149.154
C06199=1194.176,-73.385,-40.464,179.440,5.597,149.154
C06200=1194.171,-73.135,-40.476,179.443,5.596,149.153
C06201=1194.166,-72.885,-40.486,179.445,5.597,149.152
C06202=1194.161,-72.636,-40.497,179.447,5.598,149.152
C06203=1194.156,-72.386,-40.508,179.449,5.597,149.151
C06204=1194.150,-72.137,-40.519,179.452,5.598,149.150
C06205=1194.145,-71.886,-40.530,179.454,5.599,149.150
C06206=1194.140,-71.637,-40.541,179.456,5.598,149.149
C06207=1194.135,-71.387,-40.551,179.459,5.599,149.148
C06208=1194.129,-71.137,-40.563,179.461,5.598,149.148
C06209=1194.124,-70.888,-40.574,179.463,5.599,149.147
C06210=1194.119,-70.638,-40.585,179.466,5.600,149.147
C06211=1194.114,-70.388,-40.596,179.468,5.599,149.146
C06212=1194.108,-70.139,-40.607,179.471,5.600,149.145
C06213=1194.103,-69.889,-40.618,179.473,5.600,149.145
C06214=1194.099,-69.639,-40.629,179.475,5.600,149.144
C06215=1194.093,-69.390,-40.640,179.478,5.600,149.143
C06216=1194.088,-69.140,-40.651,179.480,5.600,149.143
C06217=1194.083,-68.890,-40.662,179.482,5.601,149.142
C06218=1194.077,-68.641,-40.673,179.485,5.601,149.141
C06219=1194.072,-68.391,-40.685,179.487,5.601,149.141
C06220=1194.067,-68.140,-40.695,179.489,5.601,149.140
C06221=1194.062,-67.892,-40.706,179.492,5.602,149.140
C06222=1194.056,-67.642,-40.718,179.494,5.602,149.139
C06223=1194.051,-67.391,-40.729,179.496,5.602,149.138
C06224=1194.046,-67.142,-40.740,179.499,5.603,149.137
C06225=1194.041,-66.893,-40.751,179.501,5.603,149.137
C06226=1194.036,-66.643,-40.763,179.503,5.603,149.136
C06227=1194.030,-66.393,-40.773,179.505,5.603,149.136
C06228=1194.025,-66.144,-40.784,179.508,5.603,149.135
C06229=1194.020,-65.894,-40.796,179.510,5.604,149.134
C06230=1194.014,-65.644,-40.806,179.512,5.604,149.134
C06231=1194.009,-65.394,-40.818,179.515,5.604,149.133
C06232=1194.004,-65.145,-40.830,179.518,5.604,149.132
C06233=1194.000,-64.895,-40.841,179.519,5.604,149.132
C06234=1193.993,-64.645,-40.852,179.522,5.605,149.131
C06235=1193.989,-64.396,-40.863,179.525,5.605,149.130
C06236=1193.984,-64.146,-40.874,179.527,5.605,149.130
C06237=1193.978,-63.897,-40.886,179.529,5.606,149.129
C06238=1193.973,-63.646,-40.896,179.531,5.606,149.128
C06239=1193.967,-63.396,-40.908,179.534,5.606,149.128
C06240=1193.963,-63.147,-40.920,179.536,5.606,149.127
C06241=1193.957,-62.898,-40.931,179.538,5.607,149.127
C06242=1193.952,-62.648,-40.942,179.540,5.607,149.126
C06243=1193.947,-62.398,-40.953,179.543,5.607,149.125
C06244=1193.942,-62.148,-40.965,179.545,5.607,149.124
C06245=1193.936,-61.899,-40.976,179.547,5.608,149.124
C06246=1193.932,-61.649,-40.987,179.550,5.608,149.123
C06247=1193.926,-61.399,-40.999,179.552,5.608,149.123
C06248=1193.921,-61.150,-41.010,179.555,5.608,149.122
C06249=1193.915,-60.900,-41.022,179.558,5.609,149.121
C06250=1193.910,-60.650,-41.032,179.559,5.609,149.121
C06251=1193.905,-60.400,-41.044,179.562,5.609,149.120
C06252=1193.900,-60.151,-41.056,179.564,5.609,149.119
C06253=1193.895,-59.901,-41.067,179.567,5.609,149.119
C06254=1193.890,-59.652,-41.078,179.569,5.610,149.118
C06255=1193.885,-59.402,-41.090,179.571,5.610,149.117
C06256=1193.879,-59.152,-41.101,179.573,5.610,149.117
C06257=1193.875,-58.903,-41.113,179.576,5.610,149.116
C06258=1193.869,-58.653,-41.125,179.578,5.611,149.115
C06259=1193.864,-58.404,-41.136,179.580,5.611,149.115
C06260=1193.859,-58.154,-41.147,179.583,5.611,149.114
C06261=1193.854,-57.904,-41.159,179.586,5.612,149.113
C06262=1193.848,-57.654,-41.170,179.587,5.612,149.113
C06263=1193.844,-57.404,-41.181,179.590,5.612,149.112
C06264=1193.838,-57.155,-41.193,179.593,5.613,149.111
C06265=1193.833,-56.905,-41.204,179.595,5.612,149.111
C06266=1193.827,-56.655,-41.216,179.597,5.613,149.110
C06267=1193.822,-56.405,-41.228,179.600,5.614,149.110
C06268=1193.817,-56.156,-41.239,179.602,5.613,149.109
C06269=1193.812,-55.906,-41.251,179.604,5.614,149.108
C06270=1193.807,-55.656,-41.262,179.607,5.614,149.107
C06271=1193.801,-55.407,-41.274,179.609,5.614,149.107
C06272=1193.796,-55.157,-41.285,179.611,5.614,149.106
C06273=1193.791,-54.908,-41.298,179.614,5.615,149.106
C06274=1193.787,-54.658,-41.309,179.617,5.615,149.105
C06275=1193.781,-54.408,-41.321,179.618,5.615,149.104
C06276=1193.776,-54.158,-41.333,179.621,5.616,149.104
C06277=1193.771,-53.909,-41.344,179.624,5.616,149.103
C06278=1193.765,-53.660,-41.356,179.626,5.616,149.102
C06279=1193.760,-53.410,-41.367,179.628,5.617,149.102
C06280=1193.755,-53.160,-41.379,179.630,5.617,149.101
C06281=1193.750,-52.910,-41.390,179.633,5.617,149.100
C06282=1193.745,-52.660,-41.402,179.635,5.617,149.100
C06283=1193.739,-52.410,-41.414,179.638,5.618,149.099
C06284=1193.735,-52.161,-41.425,179.639,5.618,149.099
C06285=1193.730,-51.912,-41.438,179.642,5.618,149.098
C06286=1193.724,-51.662,-41.450,179.645,5.619,149.097
C06287=1193.719,-51.413,-41.460,179.647,5.618,149.096
C06288=1193.713,-51.163,-41.472,179.649,5.619,149.096
C06289=1193.708,-50.913,-41.484,179.652,5.620,149.095
C06290=1193.703,-50.663,-41.496,179.654,5.620,149.095
C06291=1193.698,-50.413,-41.507,179.656,5.620,149.094
C06292=1193.693,-50.164,-41.520,179.659,5.620,149.093
C06293=1193.688,-49.914,-41.531,179.661,5.621,149.093
C06294=1193.683,-49.644,-41.544,179.664,5.621,149.092
C06295=1193.677,-49.374,-41.557,179.666,5.621,149.091
C06296=1193.671,-49.104,-41.570,179.669,5.621,149.091
C06297=1193.665,-48.833,-41.582,179.671,5.622,149.090
C06298=1193.660,-48.584,-41.594,179.674,5.622,149.089
C06299=1193.655,-48.334,-41.606,179.676,5.622,149.088
C06300=1193.649,-48.084,-41.618,179.679,5.622,149.088
C06301=1193.645,-47.835,-41.629,179.681,5.623,149.087
C06302=1193.639,-47.586,-41.642,179.684,5.624,149.087
C06303=1193.634,-47.336,-41.654,179.686,5.623,149.086
C06304=1193.629,-47.086,-41.666,179.688,5.624,149.085
C06305=1193.624,-46.836,-41.677,179.691,5.624,149.084
C06306=1193.619,-46.587,-41.690,179.693,5.624,149.084
C06307=1193.613,-46.337,-41.702,179.695,5.625,149.083
C06308=1193.608,-46.087,-41.713,179.698,5.625,149.083
C06309=1193.604,-45.838,-41.725,179.701,5.626,149.082
C06310=1193.598,-45.588,-41.737,179.702,5.626,149.081
C06311=1193.593,-45.338,-41.749,179.705,5.626,149.081
C06312=1193.588,-45.089,-41.762,179.708,5.626,149.080
C06313=1193.583,-44.839,-41.773,179.710,5.626,149.079
C06314=1193.577,-44.589,-41.785,179.712,5.627,149.079
C06315=1193.572,-44.340,-41.798,179.714,5.627,149.078
C06316=1193.567,-44.090,-41.809,179.717,5.628,149.077
C06317=1193.561,-43.840,-41.821,179.719,5.627,149.077
C06318=1193.557,-43.591,-41.833,179.722,5.628,149.076
C06319=1193.552,-43.341,-41.845,179.725,5.628,149.075
C06320=1193.546,-43.091,-41.857,179.727,5.629,149.075
C06321=1193.541,-42.842,-41.870,179.729,5.629,149.074
C06322=1193.536,-42.592,-41.882,179.731,5.629,149.073
C06323=1193.531,-42.342,-41.894,179.734,5.630,149.073
C06324=1193.526,-42.093,-41.906,179.736,5.630,149.072
C06325=1193.520,-41.843,-41.917,179.738,5.630,149.072
C06326=1193.515,-41.594,-41.930,179.741,5.631,149.071
C06327=1193.510,-41.344,-41.942,179.744,5.631,149.070
C06328=1193.505,-41.094,-41.954,179.746,5.631,149.069
C06329=1193.499,-40.844,-41.966,179.748,5.632,149.069
C06330=1193.494,-40.595,-41.979,179.751,5.632,149.068
C06331=1193.490,-40.345,-41.990,179.753,5.632,149.068
C06332=1193.485,-40.095,-42.003,179.755,5.632,149.067
C06333=1193.480,-39.845,-42.015,179.758,5.633,149.066
C06334=1193.474,-39.596,-42.028,179.760,5.633,149.066
C06335=1193.469,-39.346,-42.040,179.763,5.634,149.065
C06336=1193.464,-39.097,-42.052,179.765,5.633,149.064
C06337=1193.458,-38.847,-42.064,179.768,5.634,149.064
C06338=1193.453,-38.598,-42.077,179.770,5.635,149.063
C06339=1193.448,-38.348,-42.089,179.772,5.635,149.062
C06340=1193.443,-38.098,-42.101,179.775,5.635,149.062
C06341=1193.437,-37.848,-42.113,179.777,5.635,149.061
C06342=1193.432,-37.599,-42.126,179.780,5.636,149.060
C06343=1193.428,-37.350,-42.137,179.781,5.636,149.060
C06344=1193.422,-37.100,-42.150,179.784,5.636,149.059
C06345=1193.418,-36.850,-42.163,179.787,5.637,149.058
C06346=1193.412,-36.600,-42.174,179.789,5.637,149.058
C06347=1193.407,-36.351,-42.187,179.792,5.638,149.057
C06348=1193.402,-36.101,-42.199,179.794,5.638,149.057
C06349=1193.397,-35.852,-42.211,179.796,5.638,149.056
C06350=1193.392,-35.602,-42.224,179.799,5.639,149.055
C06351=1193.386,-35.352,-42.236,179.802,5.639,149.054
C06352=1193.381,-35.103,-42.249,179.803,5.639,149.054
C06353=1193.376,-34.852,-42.261,179.806,5.640,149.053
C06354=1193.371,-34.603,-42.273,179.809,5.640,149.053
C06355=1193.366,-34.354,-42.286,179.811,5.640,149.052
C06356=1193.361,-34.104,-42.298,179.813,5.640,149.051
C06357=1193.355,-33.855,-42.311,179.816,5.641,149.051
C06358=1193.350,-33.605,-42.323,179.818,5.641,149.050
C06359=1193.345,-33.355,-42.335,179.821,5.642,149.049
C06360=1193.340,-33.105,-42.348,179.823,5.641,149.049
C06361=1193.335,-32.856,-42.361,179.826,5.642,149.048
C06362=1193.329,-32.606,-42.373,179.828,5.643,149.047
C06363=1193.324,-32.356,-42.386,179.830,5.643,149.047
C06364=1193.319,-32.107,-42.398,179.832,5.643,149.046
C06365=1193.314,-31.858,-42.411,179.835,5.643,149.045
C06366=1193.309,-31.607,-42.423,179.837,5.644,149.045
C06367=1193.304,-31.358,-42.436,179.840,5.645,149.044
C06368=1193.299,-31.109,-42.448,179.843,5.645,149.044
C06369=1193.294,-30.859,-42.461,179.845,5.645,149.043
C06370=1193.288,-30.609,-42.473,179.847,5.645,149.042
C06371=1193.284,-30.359,-42.486,179.850,5.646,149.042
C06372=1193.278,-30.110,-42.498,179.852,5.646,149.041
C06373=1193.273,-29.861,-42.511,179.854,5.646,149.040
C06374=1193.267,-29.610,-42.523,179.857,5.647,149.040
C06375=1193.262,-29.361,-42.536,179.860,5.647,149.039
C06376=1193.258,-29.111,-42.549,179.862,5.648,149.038
C06377=1193.252,-28.862,-42.562,179.864,5.648,149.038
C06378=1193.247,-28.612,-42.574,179.867,5.648,149.037
C06379=1193.242,-28.363,-42.587,179.869,5.648,149.036
C06380=1193.237,-28.112,-42.599,179.872,5.649,149.036
C06381=1193.232,-27.863,-42.612,179.874,5.650,149.035
C06382=1193.226,-27.613,-42.625,179.877,5.650,149.034
C06383=1193.221,-27.364,-42.637,179.879,5.650,149.034
C06384=1193.217,-27.114,-42.650,179.881,5.650,149.033
C06385=1193.212,-26.865,-42.663,179.884,5.651,149.033
C06386=1193.206,-26.616,-42.676,179.886,5.652,149.032
C06387=1193.201,-26.366,-42.688,179.889,5.652,149.031
C06388=1193.196,-26.115,-42.701,179.891,5.652,149.031
C06389=1193.191,-25.866,-42.714,179.894,5.652,149.030
C06390=1193.185,-25.617,-42.726,179.896,5.653,149.029
C06391=1193.180,-25.367,-42.739,179.899,5.654,149.029
C06392=1193.176,-25.117,-42.752,179.901,5.654,149.028
C06393=1193.170,-24.868,-42.765,179.903,5.654,149.027
C06394=1193.165,-24.618,-42.778,179.906,5.654,149.027
C06395=1193.160,-24.368,-42.791,179.908,5.655,149.026
C06396=1193.155,-24.119,-42.803,179.911,5.655,149.025
C06397=1193.149,-23.869,-42.816,179.913,5.656,149.025
C06398=1193.144,-23.600,-42.830,179.915,5.656,149.024
C06399=1193.139,-23.330,-42.844,179.918,5.656,149.023
C06400=1193.133,-23.061,-42.858,179.921,5.656,149.023
C06401=1193.128,-22.791,-42.871,179.923,5.657,149.022
C06402=1193.122,-22.541,-42.885,179.926,5.657,149.021
C06403=1193.118,-22.291,-42.898,179.929,5.658,149.021
C06404=1193.112,-22.042,-42.910,179.931,5.659,149.020
C06405=1193.107,-21.792,-42.923,179.934,5.659,149.019
C06406=1193.102,-21.542,-42.936,179.936,5.659,149.019
C06407=1193.097,-21.293,-42.949,179.938,5.659,149.018
C06408=1193.092,-21.044,-42.961,179.941,5.660,149.017
C06409=1193.087,-20.793,-42.975,179.943,5.661,149.017
C06410=1193.081,-20.544,-42.988,179.946,5.661,149.016
C06411=1193.077,-20.295,-43.001,179.949,5.662,149.015
C06412=1193.071,-20.045,-43.015,179.951,5.661,149.015
C06413=1193.066,-19.796,-43.027,179.953,5.662,149.014
C06414=1193.061,-19.546,-43.040,179.955,5.663,149.014
C06415=1193.056,-19.296,-43.053,179.958,5.663,149.013
C06416=1193.051,-19.047,-43.066,179.961,5.663,149.012
C06417=1193.046,-18.797,-43.078,179.963,5.663,149.011
C06418=1193.040,-18.547,-43.092,179.965,5.664,149.011
C06419=1193.036,-18.298,-43.105,179.968,5.664,149.010
C06420=1193.030,-18.048,-43.119,179.970,5.665,149.010
C06421=1193.025,-17.799,-43.132,179.973,5.665,149.009
C06422=1193.020,-17.549,-43.144,179.976,5.666,149.008
C06423=1193.015,-17.299,-43.158,179.977,5.666,149.008
C06424=1193.010,-17.050,-43.170,179.980,5.666,149.007
C06425=1193.005,-16.801,-43.184,179.983,5.667,149.006
C06426=1193.000,-16.551,-43.197,179.985,5.667,149.006
C06427=1192.994,-16.301,-43.210,179.988,5.668,149.005
C06428=1192.989,-16.051,-43.223,179.990,5.669,149.005
C06429=1192.984,-15.802,-43.236,179.993,5.669,149.004
C06430=1192.979,-15.552,-43.250,179.995,5.669,149.003
C06431=1192.974,-15.303,-43.263,179.997,5.669,149.002
C06432=1192.969,-15.053,-43.275,180.000,5.670,149.002
C06433=1192.964,-14.803,-43.289,-179.998,5.671,149.001
C06434=1192.959,-14.554,-43.302,-179.995,5.671,149.001
C06435=1192.954,-14.304,-43.316,-179.992,5.671,149.000
C06436=1192.948,-14.055,-43.328,-179.990,5.671,148.999
C06437=1192.943,-13.804,-43.342,-179.988,5.672,148.999
C06438=1192.938,-13.556,-43.355,-179.986,5.672,148.998
C06439=1192.932,-13.306,-43.369,-179.983,5.673,148.997
C06440=1192.928,-13.056,-43.381,-179.980,5.673,148.997
C06441=1192.922,-12.807,-43.395,-179.978,5.674,148.996
C06442=1192.918,-12.557,-43.408,-179.975,5.675,148.995
C06443=1192.912,-12.307,-43.422,-179.973,5.674,148.995
C06444=1192.908,-12.058,-43.435,-179.971,5.675,148.994
C06445=1192.902,-11.808,-43.448,-179.968,5.675,148.993
C06446=1192.897,-11.558,-43.461,-179.966,5.676,148.993
C06447=1192.892,-11.309,-43.475,-179.963,5.677,148.992
C06448=1192.887,-11.059,-43.488,-179.961,5.677,148.992
C06449=1192.882,-10.810,-43.502,-179.958,5.678,148.991
C06450=1192.877,-10.560,-43.515,-179.956,5.677,148.990
C06451=1192.871,-10.311,-43.528,-179.954,5.678,148.990
C06452=1192.867,-10.061,-43.542,-179.951,5.679,148.989
C06453=1192.861,-9.812,-43.555,-179.948,5.679,148.988
C06454=1192.857,-9.562,-43.569,-179.946,5.680,148.988
C06455=1192.851,-9.313,-43.582,-179.943,5.680,148.987
C06456=1192.847,-9.063,-43.595,-179.941,5.681,148.986
C06457=1192.841,-8.814,-43.609,-179.938,5.681,148.986
C06458=1192.836,-8.563,-43.623,-179.936,5.681,148.985
C06459=1192.831,-8.315,-43.636,-179.933,5.681,148.984
C06460=1192.826,-8.064,-43.649,-179.931,5.682,148.984
C06461=1192.821,-7.815,-43.663,-179.929,5.683,148.983
C06462=1192.816,-7.565,-43.676,-179.926,5.683,148.983
C06463=1192.811,-7.315,-43.691,-179.923,5.684,148.982
C06464=1192.806,-7.066,-43.703,-179.921,5.684,148.981
C06465=1192.801,-6.816,-43.717,-179.919,5.685,148.981
C06466=1192.796,-6.567,-43.730,-179.916,5.685,148.980
C06467=1192.791,-6.317,-43.744,-179.914,5.685,148.979
C06468=1192.785,-6.068,-43.758,-179.911,5.686,148.979
C06469=1192.781,-5.818,-43.771,-179.909,5.687,148.978
C06470=1192.775,-5.569,-43.784,-179.906,5.687,148.978
C06471=1192.770,-5.319,-43.799,-179.904,5.688,148.977
C06472=1192.765,-5.069,-43.812,-179.901,5.688,148.976
C06473=1192.760,-4.820,-43.826,-179.898,5.688,148.975
C06474=1192.755,-4.570,-43.840,-179.896,5.689,148.975
C06475=1192.750,-4.321,-43.852,-179.894,5.690,148.974
C06476=1192.745,-4.071,-43.867,-179.891,5.690,148.974
C06477=1192.739,-3.821,-43.880,-179.889,5.690,148.973
C06478=1192.735,-3.572,-43.894,-179.886,5.690,148.972
C06479=1192.730,-3.323,-43.908,-179.884,5.691,148.972
C06480=1192.724,-3.073,-43.921,-179.881,5.692,148.971
C06481=1192.720,-2.823,-43.935,-179.879,5.692,148.970
C06482=1192.715,-2.574,-43.949,-179.876,5.693,148.970
C06483=1192.709,-2.324,-43.962,-179.874,5.694,148.969
C06484=1192.704,-2.074,-43.976,-179.871,5.694,148.969
C06485=1192.699,-1.826,-43.990,-179.869,5.695,148.968
C06486=1192.694,-1.575,-44.003,-179.866,5.694,148.967
C06487=1192.689,-1.326,-44.018,-179.864,5.695,148.966
C06488=1192.683,-1.077,-44.032,-179.862,5.696,148.966
C06489=1192.679,-0.827,-44.045,-179.859,5.696,148.965
C06490=1192.674,-0.577,-44.059,-179.856,5.697,148.965
C06491=1192.668,-0.328,-44.073,-179.854,5.697,148.964
C06492=1192.663,-0.078,-44.086,-179.852,5.698,148.963
C06493=1192.659,0.172,-44.100,-179.849,5.698,148.963
C06494=1192.653,0.421,-44.114,-179.846,5.699,148.962
C06495=1192.648,0.671,-44.128,-179.844,5.699,148.961
C06496=1192.643,0.921,-44.142,-179.841,5.700,148.961
C06497=1192.637,1.170,-44.156,-179.839,5.700,148.960
C06498=1192.633,1.419,-44.169,-179.837,5.700,148.960
C06499=1192.628,1.669,-44.184,-179.834,5.701,148.959
C06500=1192.623,1.918,-44.197,-179.831,5.701,148.958
C06501=1192.617,2.168,-44.211,-179.829,5.702,148.958
C06502=1192.612,2.437,-44.227,-179.827,5.703,148.957
C06503=1192.607,2.707,-44.242,-179.824,5.703,148.956
C06504=1192.601,2.975,-44.256,-179.821,5.704,148.956
C06505=1192.595,3.245,-44.271,-179.818,5.705,148.955
C06506=1192.590,3.494,-44.286,-179.816,5.705,148.954
C06507=1192.586,3.744,-44.299,-179.813,5.705,148.954
C06508=1192.581,3.993,-44.313,-179.811,5.706,148.953
C06509=1192.576,4.242,-44.328,-179.808,5.706,148.952
C06510=1192.570,4.493,-44.341,-179.806,5.707,148.952
C06511=1192.565,4.742,-44.355,-179.803,5.707,148.951
C06512=1192.560,4.992,-44.369,-179.800,5.708,148.950
C06513=1192.555,5.241,-44.384,-179.798,5.709,148.950
C06514=1192.550,5.491,-44.398,-179.796,5.709,148.949
C06515=1192.544,5.740,-44.412,-179.793,5.710,148.949
C06516=1192.540,5.989,-44.425,-179.790,5.710,148.948
C06517=1192.535,6.239,-44.440,-179.788,5.711,148.947
C06518=1192.530,6.489,-44.454,-179.786,5.712,148.947
C06519=1192.525,6.738,-44.468,-179.783,5.712,148.946
C06520=1192.520,6.987,-44.482,-179.780,5.713,148.945
C06521=1192.515,7.237,-44.496,-179.778,5.713,148.945
C06522=1192.510,7.487,-44.511,-179.775,5.714,148.944
C06523=1192.504,7.737,-44.524,-179.773,5.714,148.944
C06524=1192.499,7.986,-44.538,-179.771,5.714,148.943
C06525=1192.494,8.236,-44.552,-179.768,5.715,148.942
C06526=1192.489,8.486,-44.567,-179.766,5.715,148.942
C06527=1192.484,8.735,-44.581,-179.763,5.716,148.941
C06528=1192.479,8.984,-44.596,-179.761,5.716,148.940
C06529=1192.474,9.233,-44.610,-179.758,5.717,148.940
C06530=1192.469,9.483,-44.624,-179.756,5.718,148.939
C06531=1192.464,9.733,-44.638,-179.753,5.718,148.939
C06532=1192.459,9.983,-44.653,-179.750,5.719,148.938
C06533=1192.454,10.232,-44.667,-179.748,5.719,148.937
C06534=1192.449,10.481,-44.681,-179.745,5.720,148.936
C06535=1192.444,10.731,-44.695,-179.743,5.721,148.936
C06536=1192.439,10.981,-44.710,-179.740,5.721,148.935
C06537=1192.434,11.230,-44.724,-179.738,5.722,148.935
C06538=1192.428,11.479,-44.738,-179.735,5.722,148.934
C06539=1192.423,11.729,-44.752,-179.733,5.723,148.933
C06540=1192.418,11.979,-44.766,-179.730,5.723,148.933
C06541=1192.414,12.228,-44.781,-179.728,5.724,148.932
C06542=1192.409,12.478,-44.796,-179.725,5.724,148.931
C06543=1192.404,12.727,-44.810,-179.723,5.725,148.931
C06544=1192.399,12.977,-44.824,-179.720,5.726,148.930
C06545=1192.393,13.226,-44.838,-179.717,5.726,148.930
C06546=1192.388,13.476,-44.852,-179.715,5.727,148.929
C06547=1192.383,13.726,-44.867,-179.713,5.728,148.928
C06548=1192.378,13.975,-44.882,-179.710,5.728,148.928
C06549=1192.373,14.225,-44.896,-179.707,5.729,148.927
C06550=1192.368,14.474,-44.911,-179.705,5.729,148.926
C06551=1192.363,14.724,-44.925,-179.703,5.730,148.926
C06552=1192.357,14.973,-44.939,-179.700,5.730,148.925
C06553=1192.353,15.222,-44.954,-179.697,5.731,148.925
C06554=1192.348,15.472,-44.968,-179.695,5.731,148.924
C06555=1192.342,15.722,-44.983,-179.692,5.732,148.923
C06556=1192.337,15.972,-44.997,-179.690,5.733,148.923
C06557=1192.333,16.221,-45.012,-179.687,5.733,148.922
C06558=1192.328,16.470,-45.027,-179.684,5.734,148.921
C06559=1192.323,16.720,-45.041,-179.682,5.735,148.921
C06560=1192.318,16.969,-45.056,-179.680,5.735,148.920
C06561=1192.313,17.219,-45.070,-179.677,5.736,148.920
C06562=1192.307,17.469,-45.085,-179.674,5.736,148.919
C06563=1192.302,17.718,-45.099,-179.672,5.737,148.918
C06564=1192.297,17.967,-45.114,-179.670,5.738,148.918
C06565=1192.292,18.217,-45.128,-179.667,5.738,148.917
C06566=1192.287,18.466,-45.142,-179.664,5.739,148.916
C06567=1192.282,18.716,-45.158,-179.662,5.739,148.916
C06568=1192.277,18.966,-45.172,-179.659,5.740,148.915
C06569=1192.272,19.215,-45.187,-179.657,5.740,148.915
C06570=1192.267,19.464,-45.202,-179.654,5.741,148.914
C06571=1192.262,19.714,-45.216,-179.652,5.742,148.913
C06572=1192.257,19.964,-45.231,-179.649,5.742,148.913
C06573=1192.252,20.213,-45.246,-179.647,5.743,148.912
C06574=1192.247,20.463,-45.260,-179.644,5.743,148.911
C06575=1192.242,20.712,-45.276,-179.642,5.744,148.911
C06576=1192.237,20.962,-45.290,-179.639,5.745,148.910
C06577=1192.232,21.211,-45.305,-179.637,5.745,148.910
C06578=1192.227,21.461,-45.319,-179.634,5.746,148.909
C06579=1192.222,21.710,-45.335,-179.632,5.747,148.908
C06580=1192.217,21.960,-45.349,-179.629,5.747,148.908
C06581=1192.212,22.210,-45.363,-179.627,5.748,148.907
C06582=1192.207,22.459,-45.378,-179.624,5.748,148.906
C06583=1192.201,22.709,-45.393,-179.622,5.749,148.906
C06584=1192.197,22.958,-45.408,-179.619,5.749,148.905
C06585=1192.192,23.208,-45.422,-179.616,5.750,148.905
C06586=1192.186,23.457,-45.438,-179.614,5.751,148.904
C06587=1192.182,23.707,-45.452,-179.612,5.751,148.903
C06588=1192.177,23.956,-45.467,-179.609,5.752,148.903
C06589=1192.171,24.206,-45.482,-179.606,5.752,148.902
C06590=1192.167,24.455,-45.497,-179.604,5.753,148.902
C06591=1192.162,24.704,-45.512,-179.602,5.754,148.901
C06592=1192.156,24.954,-45.527,-179.599,5.754,148.900
C06593=1192.152,25.203,-45.542,-179.596,5.755,148.900
C06594=1192.147,25.453,-45.556,-179.594,5.756,148.899
C06595=1192.141,25.702,-45.572,-179.591,5.756,148.898
C06596=1192.136,25.952,-45.586,-179.589,5.757,148.898
C06597=1192.131,26.201,-45.602,-179.586,5.757,148.897
C06598=1192.126,26.450,-45.617,-179.583,5.759,148.897
C06599=1192.121,26.700,-45.631,-179.581,5.759,148.896
C06600=1192.116,26.950,-45.647,-179.578,5.760,148.895
C06601=1192.112,27.200,-45.661,-179.576,5.761,148.895
C06602=1192.106,27.449,-45.677,-179.573,5.761,148.894
C06603=1192.101,27.698,-45.692,-179.571,5.762,148.894
C06604=1192.096,27.948,-45.707,-179.568,5.762,148.893
C06605=1192.091,28.198,-45.722,-179.566,5.763,148.892
C06606=1192.086,28.466,-45.737,-179.563,5.764,148.892
C06607=1192.080,28.735,-45.754,-179.561,5.764,148.891
C06608=1192.075,29.004,-45.771,-179.557,5.765,148.890
C06609=1192.069,29.273,-45.786,-179.555,5.766,148.890
C06610=1192.064,29.522,-45.802,-179.552,5.766,148.889
C06611=1192.059,29.771,-45.817,-179.549,5.767,148.888
C06612=1192.054,30.021,-45.831,-179.547,5.768,148.888
C06613=1192.049,30.270,-45.847,-179.545,5.768,148.887
C06614=1192.044,30.519,-45.862,-179.542,5.769,148.887
C06615=1192.040,30.770,-45.878,-179.540,5.770,148.886
C06616=1192.035,31.019,-45.892,-179.537,5.770,148.885
C06617=1192.029,31.269,-45.908,-179.534,5.771,148.885
C06618=1192.025,31.518,-45.923,-179.532,5.771,148.884
C06619=1192.019,31.767,-45.938,-179.530,5.772,148.884
C06620=1192.015,32.016,-45.953,-179.526,5.773,148.883
C06621=1192.009,32.266,-45.968,-179.524,5.774,148.882
C06622=1192.004,32.516,-45.984,-179.522,5.775,148.882
C06623=1191.999,32.765,-45.999,-179.519,5.775,148.881
C06624=1191.994,33.015,-46.015,-179.516,5.776,148.880
C06625=1191.989,33.264,-46.030,-179.514,5.776,148.880
C06626=1191.984,33.513,-46.045,-179.512,5.777,148.879
C06627=1191.979,33.763,-46.059,-179.509,5.778,148.879
C06628=1191.974,34.013,-46.075,-179.506,5.778,148.878
C06629=1191.970,34.262,-46.090,-179.504,5.779,148.878
C06630=1191.964,34.512,-46.106,-179.501,5.780,148.877
C06631=1191.959,34.761,-46.122,-179.498,5.781,148.876
C06632=1191.954,35.010,-46.137,-179.496,5.781,148.876
C06633=1191.949,35.260,-46.153,-179.493,5.782,148.875
C06634=1191.945,35.509,-46.168,-179.491,5.783,148.874
C06635=1191.939,35.759,-46.183,-179.488,5.783,148.874
C06636=1191.934,36.008,-46.199,-179.486,5.784,148.873
C06637=1191.929,36.258,-46.213,-179.483,5.785,148.873
C06638=1191.924,36.508,-46.229,-179.481,5.785,148.872
C06639=1191.919,36.757,-46.245,-179.479,5.786,148.871
C06640=1191.914,37.006,-46.260,-179.476,5.787,148.871
C06641=1191.909,37.256,-46.275,-179.473,5.788,148.870
C06642=1191.904,37.506,-46.291,-179.470,5.788,148.869
C06643=1191.899,37.755,-46.306,-179.468,5.789,148.869
C06644=1191.894,38.004,-46.322,-179.465,5.790,148.868
C06645=1191.889,38.254,-46.337,-179.463,5.790,148.868
C06646=1191.885,38.504,-46.353,-179.460,5.791,148.867
C06647=1191.879,38.753,-46.368,-179.458,5.792,148.867
C06648=1191.874,39.002,-46.384,-179.455,5.792,148.866
C06649=1191.869,39.252,-46.399,-179.453,5.793,148.865
C06650=1191.864,39.502,-46.415,-179.450,5.794,148.865
C06651=1191.859,39.750,-46.431,-179.447,5.795,148.864
C06652=1191.854,40.000,-46.447,-179.445,5.796,148.863
C06653=1191.849,40.249,-46.462,-179.442,5.796,148.863
C06654=1191.845,40.499,-46.478,-179.440,5.797,148.862
C06655=1191.839,40.748,-46.493,-179.437,5.797,148.862
C06656=1191.834,40.998,-46.509,-179.435,5.798,148.861
C06657=1191.830,41.248,-46.524,-179.432,5.799,148.860
C06658=1191.824,41.497,-46.540,-179.429,5.800,148.860
C06659=1191.819,41.746,-46.555,-179.427,5.801,148.859
C06660=1191.814,41.995,-46.572,-179.424,5.802,148.859
C06661=1191.810,42.245,-46.587,-179.422,5.802,148.858
C06662=1191.804,42.494,-46.603,-179.419,5.803,148.858
C06663=1191.799,42.744,-46.618,-179.417,5.803,148.857
C06664=1191.794,42.994,-46.634,-179.414,5.804,148.856
C06665=1191.789,43.243,-46.650,-179.412,5.805,148.856
C06666=1191.785,43.492,-46.665,-179.409,5.806,148.855
C06667=1191.780,43.742,-46.681,-179.406,5.807,148.854
C06668=1191.774,43.991,-46.697,-179.404,5.807,148.854
C06669=1191.769,44.241,-46.712,-179.401,5.808,148.853
C06670=1191.764,44.491,-46.728,-179.399,5.809,148.853
C06671=1191.759,44.740,-46.745,-179.396,5.809,148.852
C06672=1191.754,44.989,-46.760,-179.394,5.810,148.852
C06673=1191.750,45.239,-46.776,-179.391,5.811,148.851
C06674=1191.744,45.488,-46.791,-179.388,5.812,148.850
C06675=1191.740,45.738,-46.808,-179.386,5.813,148.850
C06676=1191.734,45.987,-46.824,-179.383,5.813,148.849
C06677=1191.729,46.236,-46.839,-179.381,5.814,148.848
C06678=1191.725,46.486,-46.856,-179.379,5.815,148.848
C06679=1191.720,46.735,-46.871,-179.375,5.816,148.847
C06680=1191.714,46.984,-46.886,-179.373,5.817,148.847
C06681=1191.710,47.234,-46.903,-179.371,5.817,148.846
C06682=1191.705,47.483,-46.919,-179.368,5.818,148.846
C06683=1191.700,47.733,-46.935,-179.365,5.819,148.845
C06684=1191.695,47.982,-46.951,-179.363,5.819,148.844
C06685=1191.690,48.232,-46.967,-179.360,5.820,148.844
C06686=1191.685,48.482,-46.982,-179.357,5.821,148.843
C06687=1191.679,48.730,-46.999,-179.355,5.822,148.843
C06688=1191.675,48.981,-47.015,-179.352,5.823,148.842
C06689=1191.669,49.230,-47.030,-179.350,5.823,148.841
C06690=1191.665,49.479,-47.047,-179.348,5.824,148.841
C06691=1191.660,49.729,-47.062,-179.344,5.825,148.840
C06692=1191.656,49.978,-47.079,-179.342,5.826,148.840
C06693=1191.650,50.227,-47.094,-179.340,5.827,148.839
C06694=1191.645,50.476,-47.110,-179.337,5.827,148.838
C06695=1191.640,50.726,-47.126,-179.334,5.828,148.838
C06696=1191.635,50.976,-47.142,-179.332,5.829,148.837
C06697=1191.631,51.225,-47.159,-179.329,5.830,148.837
C06698=1191.625,51.475,-47.174,-179.326,5.831,148.836
C06699=1191.621,51.724,-47.191,-179.324,5.832,148.836
C06700=1191.615,51.974,-47.207,-179.322,5.832,148.835
C06701=1191.611,52.223,-47.223,-179.319,5.833,148.834
C06702=1191.605,52.472,-47.239,-179.316,5.834,148.834
C06703=1191.601,52.722,-47.255,-179.314,5.835,148.833
C06704=1191.596,52.971,-47.272,-179.311,5.835,148.832
C06705=1191.591,53.221,-47.288,-179.309,5.836,148.832
C06706=1191.585,53.470,-47.305,-179.306,5.837,148.831
C06707=1191.581,53.720,-47.321,-179.304,5.837,148.831
C06708=1191.575,53.969,-47.337,-179.301,5.839,148.830
C06709=1191.571,54.219,-47.353,-179.298,5.840,148.830
C06710=1191.565,54.487,-47.371,-179.296,5.840,148.829
C06711=1191.560,54.755,-47.388,-179.292,5.841,148.828
C06712=1191.555,55.024,-47.405,-179.290,5.842,148.828
C06713=1191.550,55.292,-47.423,-179.288,5.843,148.827
C06714=1191.544,55.542,-47.438,-179.284,5.844,148.826
C06715=1191.539,55.791,-47.456,-179.282,5.845,148.826
C06716=1191.535,56.041,-47.472,-179.280,5.846,148.825
C06717=1191.529,56.290,-47.488,-179.277,5.846,148.825
C06718=1191.525,56.540,-47.504,-179.275,5.847,148.824
C06719=1191.520,56.789,-47.521,-179.272,5.848,148.824
C06720=1191.515,57.039,-47.537,-179.269,5.849,148.823
C06721=1191.510,57.287,-47.553,-179.267,5.850,148.822
C06722=1191.505,57.537,-47.570,-179.264,5.850,148.822
C06723=1191.499,57.787,-47.586,-179.261,5.852,148.821
C06724=1191.495,58.036,-47.603,-179.259,5.853,148.821
C06725=1191.490,58.285,-47.619,-179.256,5.853,148.820
C06726=1191.485,58.534,-47.636,-179.253,5.854,148.819
C06727=1191.480,58.785,-47.651,-179.251,5.855,148.819
C06728=1191.474,59.034,-47.668,-179.248,5.856,148.818
C06729=1191.470,59.283,-47.685,-179.246,5.857,148.818
C06730=1191.465,59.532,-47.701,-179.243,5.857,148.817
C06731=1191.460,59.782,-47.717,-179.241,5.858,148.816
C06732=1191.456,60.031,-47.734,-179.238,5.860,148.816
C06733=1191.450,60.281,-47.751,-179.235,5.860,148.815
C06734=1191.445,60.530,-47.768,-179.233,5.861,148.815
C06735=1191.440,60.779,-47.784,-179.231,5.861,148.814
C06736=1191.435,61.029,-47.800,-179.227,5.863,148.814
C06737=1191.430,61.279,-47.817,-179.225,5.864,148.813
C06738=1191.425,61.528,-47.833,-179.223,5.864,148.813
C06739=1191.421,61.777,-47.850,-179.220,5.865,148.812
C06740=1191.416,62.026,-47.867,-179.218,5.866,148.811
C06741=1191.410,62.276,-47.884,-179.215,5.867,148.811
C06742=1191.406,62.525,-47.900,-179.212,5.868,148.810
C06743=1191.401,62.774,-47.916,-179.210,5.868,148.810
C06744=1191.395,63.024,-47.933,-179.207,5.869,148.809
C06745=1191.391,63.274,-47.950,-179.204,5.871,148.809
C06746=1191.386,63.523,-47.966,-179.202,5.871,148.808
C06747=1191.381,63.772,-47.983,-179.199,5.872,148.807
C06748=1191.376,64.022,-48.000,-179.197,5.873,148.807
C06749=1191.371,64.271,-48.016,-179.194,5.874,148.806
C06750=1191.367,64.520,-48.033,-179.191,5.875,148.806
C06751=1191.361,64.770,-48.050,-179.189,5.875,148.805
C06752=1191.357,65.019,-48.067,-179.186,5.877,148.804
C06753=1191.352,65.268,-48.083,-179.184,5.878,148.804
C06754=1191.347,65.518,-48.101,-179.181,5.878,148.803
C06755=1191.342,65.767,-48.117,-179.178,5.879,148.803
C06756=1191.336,66.017,-48.134,-179.176,5.881,148.802
C06757=1191.332,66.266,-48.151,-179.173,5.881,148.802
C06758=1191.327,66.515,-48.167,-179.171,5.882,148.801
C06759=1191.321,66.765,-48.184,-179.168,5.882,148.800
C06760=1191.317,67.014,-48.201,-179.165,5.884,148.800
C06761=1191.312,67.264,-48.218,-179.163,5.885,148.799
C06762=1191.307,67.513,-48.235,-179.160,5.885,148.799
C06763=1191.302,67.762,-48.251,-179.158,5.886,148.798
C06764=1191.297,68.012,-48.268,-179.155,5.888,148.798
C06765=1191.292,68.261,-48.285,-179.152,5.888,148.797
C06766=1191.287,68.511,-48.302,-179.150,5.889,148.797
C06767=1191.282,68.760,-48.319,-179.147,5.890,148.796
C06768=1191.278,69.009,-48.336,-179.145,5.891,148.795
C06769=1191.273,69.259,-48.353,-179.142,5.892,148.795
C06770=1191.268,69.508,-48.370,-179.140,5.892,148.794
C06771=1191.262,69.757,-48.387,-179.137,5.894,148.794
C06772=1191.258,70.007,-48.404,-179.134,5.895,148.793
C06773=1191.253,70.256,-48.421,-179.132,5.895,148.793
C06774=1191.248,70.506,-48.438,-179.129,5.897,148.792
C06775=1191.243,70.754,-48.455,-179.127,5.898,148.792
C06776=1191.238,71.004,-48.472,-179.124,5.898,148.791
C06777=1191.233,71.254,-48.489,-179.121,5.900,148.790
C06778=1191.229,71.503,-48.506,-179.119,5.901,148.790
C06779=1191.223,71.753,-48.523,-179.116,5.901,148.789
C06780=1191.219,72.001,-48.540,-179.114,5.902,148.789
C06781=1191.213,72.251,-48.557,-179.111,5.903,148.788
C06782=1191.209,72.500,-48.574,-179.108,5.904,148.787
C06783=1191.204,72.750,-48.591,-179.106,5.905,148.787
C06784=1191.200,72.999,-48.609,-179.103,5.906,148.786
C06785=1191.194,73.248,-48.626,-179.101,5.907,148.786
C06786=1191.189,73.498,-48.642,-179.098,5.908,148.785
C06787=1191.184,73.747,-48.659,-179.095,5.909,148.785
C06788=1191.179,73.997,-48.677,-179.093,5.910,148.784
C06789=1191.175,74.246,-48.694,-179.090,5.910,148.783
C06790=1191.169,74.496,-48.711,-179.087,5.912,148.783
C06791=1191.165,74.744,-48.728,-179.085,5.913,148.782
C06792=1191.159,74.994,-48.746,-179.083,5.914,148.782
C06793=1191.154,75.244,-48.763,-179.080,5.914,148.781
C06794=1191.150,75.493,-48.780,-179.077,5.916,148.781
C06795=1191.145,75.742,-48.798,-179.075,5.916,148.780
C06796=1191.140,75.992,-48.814,-179.072,5.917,148.780
C06797=1191.135,76.241,-48.832,-179.069,5.919,148.779
C06798=1191.130,76.491,-48.849,-179.067,5.919,148.778
C06799=1191.125,76.739,-48.867,-179.064,5.920,148.778
C06800=1191.120,76.989,-48.884,-179.061,5.921,148.777
C06801=1191.115,77.239,-48.901,-179.059,5.922,148.777
C06802=1191.111,77.487,-48.918,-179.056,5.923,148.776
C06803=1191.106,77.737,-48.936,-179.053,5.924,148.776
C06804=1191.101,77.986,-48.954,-179.051,5.925,148.775
C06805=1191.096,78.236,-48.970,-179.048,5.926,148.775
C06806=1191.091,78.485,-48.988,-179.046,5.927,148.774
C06807=1191.086,78.735,-49.006,-179.043,5.928,148.773
C06808=1191.082,78.984,-49.023,-179.041,5.929,148.773
C06809=1191.076,79.233,-49.040,-179.038,5.930,148.772
C06810=1191.071,79.482,-49.058,-179.036,5.931,148.772
C06811=1191.066,79.732,-49.075,-179.032,5.933,148.771
C06812=1191.062,79.981,-49.092,-179.030,5.933,148.771
C06813=1191.057,80.230,-49.110,-179.028,5.934,148.770
C06814=1191.051,80.499,-49.129,-179.024,5.935,148.770
C06815=1191.046,80.768,-49.148,-179.022,5.936,148.769
C06816=1191.040,81.036,-49.166,-179.019,5.938,148.769
C06817=1191.036,81.304,-49.185,-179.016,5.938,148.768
C06818=1191.031,81.553,-49.202,-179.013,5.940,148.767
C06819=1191.026,81.803,-49.220,-179.011,5.940,148.767
C06820=1191.021,82.052,-49.238,-179.009,5.941,148.766
C06821=1191.015,82.302,-49.255,-179.006,5.943,148.766
C06822=1191.011,82.550,-49.273,-179.003,5.943,148.765
C06823=1191.006,82.800,-49.290,-179.000,5.945,148.765
C06824=1191.001,83.049,-49.308,-178.998,5.946,148.764
C06825=1190.996,83.299,-49.326,-178.996,5.946,148.764
C06826=1190.991,83.548,-49.343,-178.993,5.948,148.763
C06827=1190.987,83.797,-49.361,-178.990,5.949,148.762
C06828=1190.982,84.046,-49.379,-178.988,5.949,148.762
C06829=1190.977,84.296,-49.396,-178.985,5.951,148.761
C06830=1190.972,84.545,-49.414,-178.982,5.952,148.761
C06831=1190.967,84.795,-49.432,-178.980,5.953,148.760
C06832=1190.962,85.044,-49.450,-178.977,5.954,148.760
C06833=1190.958,85.293,-49.467,-178.974,5.954,148.759
C06834=1190.953,85.542,-49.485,-178.972,5.956,148.759
C06835=1190.948,85.792,-49.503,-178.969,5.957,148.758
C06836=1190.942,86.041,-49.520,-178.967,5.958,148.758
C06837=1190.938,86.291,-49.538,-178.964,5.959,148.757
C06838=1190.933,86.540,-49.556,-178.962,5.960,148.756
C06839=1190.928,86.789,-49.574,-178.958,5.961,148.756
C06840=1190.923,87.038,-49.592,-178.956,5.962,148.755
C06841=1190.918,87.288,-49.609,-178.954,5.963,148.755
C06842=1190.913,87.538,-49.627,-178.951,5.964,148.754
C06843=1190.909,87.787,-49.645,-178.948,5.965,148.754
C06844=1190.904,88.036,-49.663,-178.946,5.967,148.753
C06845=1190.899,88.285,-49.681,-178.943,5.967,148.753
C06846=1190.894,88.535,-49.698,-178.941,5.968,148.752
C06847=1190.889,88.784,-49.716,-178.938,5.970,148.752
C06848=1190.884,89.033,-49.734,-178.936,5.970,148.751
C06849=1190.879,89.282,-49.752,-178.932,5.972,148.750
C06850=1190.874,89.532,-49.770,-178.930,5.973,148.750
C06851=1190.870,89.781,-49.788,-178.928,5.973,148.749
C06852=1190.865,90.030,-49.806,-178.925,5.975,148.749
C06853=1190.860,90.279,-49.824,-178.922,5.976,148.748
C06854=1190.855,90.529,-49.842,-178.920,5.977,148.748
C06855=1190.850,90.779,-49.859,-178.917,5.978,148.747
C06856=1190.845,91.028,-49.877,-178.914,5.980,148.747
C06857=1190.840,91.277,-49.895,-178.912,5.980,148.746
C06858=1190.835,91.526,-49.913,-178.909,5.981,148.746
C06859=1190.831,91.775,-49.931,-178.906,5.982,148.745
C06860=1190.826,92.025,-49.949,-178.904,5.983,148.745
C06861=1190.821,92.274,-49.968,-178.901,5.985,148.744
C06862=1190.816,92.524,-49.986,-178.899,5.986,148.744
C06863=1190.811,92.773,-50.004,-178.896,5.986,148.743
C06864=1190.806,93.022,-50.022,-178.893,5.988,148.743
C06865=1190.801,93.271,-50.040,-178.891,5.989,148.742
C06866=1190.796,93.521,-50.058,-178.888,5.990,148.742
C06867=1190.791,93.770,-50.076,-178.885,5.991,148.741
C06868=1190.787,94.020,-50.094,-178.883,5.993,148.740
C06869=1190.782,94.269,-50.112,-178.880,5.993,148.740
C06870=1190.777,94.517,-50.131,-178.877,5.995,148.739
C06871=1190.772,94.767,-50.149,-178.875,5.995,148.739
C06872=1190.767,95.016,-50.167,-178.873,5.996,148.738
C06873=1190.763,95.266,-50.185,-178.869,5.998,148.738
C06874=1190.757,95.515,-50.204,-178.867,5.999,148.737
C06875=1190.753,95.764,-50.222,-178.864,6.000,148.737
C06876=1190.748,96.014,-50.240,-178.862,6.001,148.736
C06877=1190.743,96.263,-50.258,-178.859,6.003,148.736
C06878=1190.738,96.513,-50.276,-178.857,6.003,148.735
C06879=1190.734,96.761,-50.295,-178.854,6.005,148.735
C06880=1190.728,97.011,-50.314,-178.851,6.006,148.734
C06881=1190.723,97.260,-50.332,-178.849,6.006,148.734
C06882=1190.718,97.509,-50.350,-178.846,6.008,148.733
C06883=1190.714,97.759,-50.368,-178.844,6.009,148.733
C06884=1190.709,98.007,-50.387,-178.841,6.010,148.732
C06885=1190.704,98.257,-50.405,-178.839,6.011,148.732
C06886=1190.699,98.506,-50.423,-178.835,6.012,148.731
C06887=1190.695,98.756,-50.442,-178.833,6.013,148.730
C06888=1190.690,99.004,-50.460,-178.830,6.015,148.730
C06889=1190.685,99.254,-50.478,-178.828,6.016,148.729
C06890=1190.679,99.503,-50.497,-178.825,6.017,148.729
C06891=1190.675,99.753,-50.515,-178.823,6.018,148.728
C06892=1190.670,100.002,-50.534,-178.820,6.020,148.728
C06893=1190.666,100.251,-50.552,-178.817,6.020,148.727
C06894=1190.661,100.501,-50.571,-178.815,6.022,148.727
C06895=1190.656,100.750,-50.589,-178.812,6.023,148.726
C06896=1190.651,100.999,-50.607,-178.810,6.023,148.726
C06897=1190.645,101.248,-50.626,-178.807,6.025,148.725
C06898=1190.641,101.498,-50.644,-178.804,6.026,148.725
C06899=1190.636,101.747,-50.663,-178.801,6.027,148.724
C06900=1190.632,101.996,-50.681,-178.799,6.028,148.724
C06901=1190.627,102.245,-50.701,-178.796,6.030,148.723
C06902=1190.622,102.495,-50.719,-178.794,6.030,148.723
C06903=1190.617,102.744,-50.737,-178.791,6.032,148.722
C06904=1190.612,102.993,-50.756,-178.788,6.033,148.722
C06905=1190.607,103.242,-50.774,-178.786,6.034,148.721
C06906=1190.603,103.491,-50.793,-178.783,6.035,148.721
C06907=1190.598,103.741,-50.812,-178.780,6.037,148.720
C06908=1190.593,103.990,-50.830,-178.778,6.037,148.720
C06909=1190.587,104.239,-50.849,-178.775,6.039,148.719
C06910=1190.583,104.489,-50.867,-178.773,6.040,148.719
C06911=1190.578,104.738,-50.886,-178.770,6.041,148.718
C06912=1190.573,104.987,-50.905,-178.768,6.042,148.718
C06913=1190.569,105.236,-50.924,-178.764,6.044,148.717
C06914=1190.563,105.486,-50.942,-178.762,6.045,148.717
C06915=1190.559,105.735,-50.961,-178.759,6.046,148.716
C06916=1190.554,105.984,-50.979,-178.757,6.047,148.716
C06917=1190.549,106.233,-50.999,-178.754,6.049,148.715
C06918=1190.544,106.502,-51.019,-178.751,6.050,148.715
C06919=1190.539,106.770,-51.039,-178.749,6.051,148.714
C06920=1190.533,107.039,-51.059,-178.746,6.052,148.713
C06921=1190.529,107.307,-51.080,-178.743,6.054,148.713
C06922=1190.523,107.556,-51.098,-178.741,6.055,148.712
C06923=1190.519,107.805,-51.117,-178.737,6.056,148.712
C06924=1190.514,108.055,-51.136,-178.735,6.057,148.711
C06925=1190.509,108.304,-51.155,-178.732,6.059,148.711
C06926=1190.504,108.553,-51.174,-178.730,6.059,148.710
C06927=1190.499,108.803,-51.192,-178.727,6.061,148.710
C06928=1190.495,109.052,-51.212,-178.725,6.062,148.709
C06929=1190.490,109.301,-51.231,-178.722,6.063,148.709
C06930=1190.485,109.551,-51.250,-178.720,6.064,148.708
C06931=1190.480,109.799,-51.268,-178.717,6.066,148.708
C06932=1190.475,110.048,-51.288,-178.714,6.067,148.707
C06933=1190.471,110.298,-51.306,-178.711,6.068,148.707
C06934=1190.465,110.547,-51.325,-178.709,6.070,148.706
C06935=1190.461,110.796,-51.344,-178.706,6.071,148.706
C06936=1190.456,111.046,-51.363,-178.703,6.072,148.705
C06937=1190.452,111.295,-51.382,-178.701,6.073,148.705
C06938=1190.446,111.544,-51.401,-178.698,6.074,148.704
C06939=1190.442,111.793,-51.421,-178.696,6.075,148.704
C06940=1190.437,112.043,-51.439,-178.693,6.077,148.703
C06941=1190.432,112.292,-51.458,-178.690,6.078,148.703
C06942=1190.427,112.541,-51.477,-178.688,6.079,148.702
C06943=1190.423,112.790,-51.497,-178.685,6.081,148.702
C06944=1190.417,113.040,-51.515,-178.682,6.082,148.701
C06945=1190.413,113.289,-51.534,-178.680,6.083,148.701
C06946=1190.408,113.538,-51.554,-178.677,6.084,148.700
C06947=1190.404,113.787,-51.573,-178.674,6.086,148.700
C06948=1190.398,114.036,-51.592,-178.672,6.086,148.699
C06949=1190.394,114.286,-51.612,-178.669,6.088,148.699
C06950=1190.389,114.535,-51.630,-178.667,6.089,148.699
C06951=1190.384,114.784,-51.649,-178.664,6.090,148.698
C06952=1190.379,115.033,-51.669,-178.661,6.092,148.697
C06953=1190.375,115.282,-51.688,-178.659,6.093,148.697
C06954=1190.369,115.531,-51.707,-178.656,6.094,148.696
C06955=1190.364,115.781,-51.727,-178.654,6.095,148.696
C06956=1190.360,116.029,-51.745,-178.650,6.097,148.695
C06957=1190.355,116.279,-51.765,-178.648,6.098,148.695
C06958=1190.350,116.529,-51.785,-178.646,6.099,148.695
C06959=1190.345,116.777,-51.804,-178.642,6.101,148.694
C06960=1190.341,117.027,-51.822,-178.640,6.102,148.694
C06961=1190.335,117.276,-51.842,-178.638,6.104,148.693
C06962=1190.331,117.526,-51.861,-178.635,6.104,148.693
C06963=1190.326,117.774,-51.880,-178.632,6.106,148.692
C06964=1190.321,118.024,-51.900,-178.630,6.108,148.692
C06965=1190.316,118.273,-51.919,-178.627,6.108,148.691
C06966=1190.311,118.522,-51.939,-178.624,6.110,148.691
C06967=1190.306,118.772,-51.958,-178.622,6.111,148.690
C06968=1190.302,119.020,-51.977,-178.619,6.112,148.690
C06969=1190.297,119.269,-51.997,-178.616,6.114,148.689
C06970=1190.293,119.519,-52.017,-178.614,6.115,148.689
C06971=1190.287,119.768,-52.036,-178.611,6.116,148.688
C06972=1190.283,120.017,-52.055,-178.609,6.117,148.688
C06973=1190.278,120.266,-52.075,-178.606,6.119,148.687
C06974=1190.273,120.516,-52.094,-178.603,6.120,148.687
C06975=1190.268,120.765,-52.114,-178.601,6.121,148.686
C06976=1190.263,121.014,-52.133,-178.598,6.123,148.686
C06977=1190.258,121.264,-52.153,-178.596,6.124,148.685
C06978=1190.254,121.513,-52.172,-178.593,6.125,148.685
C06979=1190.249,121.761,-52.192,-178.590,6.127,148.684
C06980=1190.245,122.011,-52.212,-178.588,6.128,148.684
C06981=1190.240,122.260,-52.231,-178.585,6.130,148.684
C06982=1190.234,122.509,-52.251,-178.582,6.130,148.683
C06983=1190.230,122.759,-52.270,-178.580,6.132,148.683
C06984=1190.225,123.008,-52.290,-178.577,6.134,148.682
C06985=1190.221,123.256,-52.309,-178.574,6.134,148.681
C06986=1190.216,123.506,-52.329,-178.572,6.136,148.681
C06987=1190.211,123.755,-52.349,-178.569,6.138,148.681
C06988=1190.206,124.004,-52.368,-178.566,6.138,148.680
C06989=1190.201,124.253,-52.388,-178.564,6.140,148.680
C06990=1190.197,124.503,-52.408,-178.561,6.141,148.679
C06991=1190.192,124.752,-52.428,-178.558,6.142,148.679
C06992=1190.187,125.001,-52.447,-178.556,6.144,148.678
C06993=1190.182,125.250,-52.467,-178.553,6.145,148.678
C06994=1190.177,125.500,-52.487,-178.551,6.147,148.677
C06995=1190.172,125.748,-52.506,-178.548,6.148,148.677
C06996=1190.168,125.997,-52.527,-178.545,6.149,148.676
C06997=1190.163,126.247,-52.546,-178.543,6.151,148.676
C06998=1190.158,126.497,-52.566,-178.540,6.152,148.675
C06999=1190.153,126.745,-52.586,-178.537,6.153,148.675
C07000=1190.148,126.994,-52.605,-178.535,6.155,148.675
C07001=1190.144,127.244,-52.625,-178.532,6.156,148.674
C07002=1190.139,127.493,-52.646,-178.529,6.157,148.674
C07003=1190.134,127.742,-52.665,-178.527,6.159,148.673
C07004=1190.129,127.991,-52.684,-178.524,6.160,148.673
C07005=1190.125,128.240,-52.705,-178.521,6.162,148.672
C07006=1190.120,128.490,-52.724,-178.519,6.163,148.672
C07007=1190.115,128.739,-52.745,-178.517,6.164,148.671
C07008=1190.110,128.988,-52.764,-178.513,6.166,148.671
C07009=1190.106,129.237,-52.785,-178.511,6.167,148.670
C07010=1190.101,129.486,-52.804,-178.509,6.168,148.670
C07011=1190.097,129.735,-52.825,-178.505,6.170,148.669
C07012=1190.092,129.985,-52.844,-178.503,6.171,148.669
C07013=1190.087,130.233,-52.864,-178.501,6.172,148.669
C07014=1190.082,130.482,-52.884,-178.497,6.174,148.668
C07015=1190.078,130.731,-52.904,-178.495,6.176,148.668
C07016=1190.073,130.981,-52.924,-178.493,6.177,148.667
C07017=1190.068,131.230,-52.944,-178.490,6.178,148.667
C07018=1190.062,131.479,-52.964,-178.487,6.180,148.666
C07019=1190.058,131.728,-52.985,-178.485,6.181,148.666
C07020=1190.053,131.978,-53.004,-178.482,6.182,148.665
C07021=1190.049,132.227,-53.025,-178.479,6.184,148.665
C07022=1190.043,132.496,-53.046,-178.476,6.186,148.664
C07023=1190.038,132.764,-53.068,-178.473,6.187,148.664
C07024=1190.033,133.033,-53.090,-178.471,6.188,148.663
C07025=1190.028,133.301,-53.111,-178.468,6.190,148.663
C07026=1190.023,133.550,-53.131,-178.465,6.191,148.662
C07027=1190.019,133.799,-53.152,-178.462,6.193,148.662
C07028=1190.014,134.049,-53.172,-178.460,6.194,148.661
C07029=1190.009,134.298,-53.192,-178.457,6.196,148.661
C07030=1190.005,134.547,-53.213,-178.454,6.197,148.660
C07031=1189.999,134.796,-53.232,-178.452,6.198,148.660
C07032=1189.995,135.045,-53.252,-178.449,6.200,148.660
C07033=1189.990,135.294,-53.273,-178.447,6.201,148.659
C07034=1189.985,135.544,-53.293,-178.444,6.203,148.659
C07035=1189.980,135.792,-53.313,-178.441,6.204,148.658
C07036=1189.976,136.041,-53.334,-178.439,6.206,148.658
C07037=1189.971,136.291,-53.355,-178.436,6.207,148.658
C07038=1189.966,136.540,-53.374,-178.433,6.208,148.657
C07039=1189.962,136.789,-53.395,-178.431,6.210,148.657
C07040=1189.957,137.038,-53.415,-178.428,6.211,148.656
C07041=1189.951,137.287,-53.436,-178.425,6.213,148.656
C07042=1189.947,137.536,-53.455,-178.423,6.214,148.655
C07043=1189.942,137.785,-53.476,-178.420,6.216,148.655
C07044=1189.937,138.034,-53.497,-178.417,6.217,148.654
C07045=1189.933,138.283,-53.517,-178.415,6.218,148.654
C07046=1189.928,138.532,-53.537,-178.412,6.220,148.653
C07047=1189.923,138.782,-53.558,-178.409,6.221,148.653
C07048=1189.918,139.031,-53.578,-178.407,6.223,148.653
C07049=1189.914,139.280,-53.598,-178.405,6.224,148.652
C07050=1189.909,139.529,-53.619,-178.402,6.226,148.652
C07051=1189.904,139.778,-53.640,-178.399,6.227,148.651
C07052=1189.900,140.027,-53.660,-178.397,6.228,148.651
C07053=1189.895,140.277,-53.681,-178.394,6.230,148.650
C07054=1189.890,140.526,-53.701,-178.391,6.232,148.650
C07055=1189.886,140.774,-53.722,-178.388,6.233,148.649
C07056=1189.881,141.024,-53.743,-178.386,6.234,148.649
C07057=1189.876,141.273,-53.763,-178.383,6.236,148.649
C07058=1189.871,141.523,-53.783,-178.381,6.238,148.648
C07059=1189.866,141.772,-53.804,-178.377,6.239,148.648
C07060=1189.862,142.020,-53.824,-178.375,6.240,148.647
C07061=1189.857,142.270,-53.845,-178.373,6.242,148.647
C07062=1189.852,142.519,-53.865,-178.370,6.244,148.646
C07063=1189.847,142.768,-53.886,-178.367,6.245,148.646
C07064=1189.843,143.017,-53.907,-178.365,6.246,148.645
C07065=1189.837,143.266,-53.928,-178.362,6.248,148.645
C07066=1189.833,143.515,-53.948,-178.359,6.249,148.645
C07067=1189.829,143.763,-53.969,-178.357,6.251,148.644
C07068=1189.824,144.013,-53.990,-178.354,6.252,148.644
C07069=1189.819,144.262,-54.010,-178.351,6.254,148.643
C07070=1189.815,144.512,-54.032,-178.349,6.255,148.643
C07071=1189.810,144.761,-54.052,-178.346,6.257,148.643
C07072=1189.805,145.010,-54.073,-178.344,6.258,148.642
C07073=1189.801,145.259,-54.094,-178.341,6.260,148.642
C07074=1189.795,145.508,-54.114,-178.338,6.261,148.641
C07075=1189.791,145.757,-54.135,-178.335,6.263,148.641
C07076=1189.786,146.006,-54.156,-178.333,6.265,148.640
C07077=1189.782,146.255,-54.177,-178.330,6.266,148.640
C07078=1189.777,146.504,-54.198,-178.328,6.268,148.640
C07079=1189.771,146.753,-54.219,-178.325,6.269,148.639
C07080=1189.767,147.002,-54.239,-178.322,6.271,148.639
C07081=1189.762,147.252,-54.261,-178.320,6.272,148.638
C07082=1189.758,147.500,-54.282,-178.317,6.273,148.638
C07083=1189.753,147.750,-54.303,-178.314,6.275,148.637
C07084=1189.749,147.999,-54.323,-178.312,6.277,148.637
C07085=1189.743,148.248,-54.344,-178.309,6.278,148.636
C07086=1189.738,148.497,-54.365,-178.306,6.279,148.636
C07087=1189.734,148.745,-54.386,-178.304,6.281,148.636
C07088=1189.729,148.995,-54.407,-178.301,6.283,148.635
C07089=1189.725,149.244,-54.428,-178.298,6.285,148.635
C07090=1189.720,149.493,-54.449,-178.296,6.286,148.635
C07091=1189.715,149.742,-54.470,-178.293,6.287,148.634
C07092=1189.711,149.991,-54.491,-178.290,6.289,148.634
C07093=1189.706,150.240,-54.512,-178.288,6.291,148.633
C07094=1189.701,150.489,-54.533,-178.285,6.292,148.633
C07095=1189.697,150.739,-54.554,-178.282,6.294,148.632
C07096=1189.692,150.987,-54.576,-178.280,6.295,148.632
C07097=1189.687,151.237,-54.597,-178.277,6.297,148.631
C07098=1189.682,151.486,-54.617,-178.274,6.298,148.631
C07099=1189.677,151.734,-54.639,-178.272,6.300,148.631
C07100=1189.673,151.984,-54.660,-178.269,6.302,148.630
C07101=1189.668,152.233,-54.681,-178.267,6.303,148.630
C07102=1189.664,152.482,-54.702,-178.264,6.305,148.630
C07103=1189.658,152.731,-54.723,-178.261,6.306,148.629
C07104=1189.653,152.980,-54.745,-178.258,6.308,148.629
C07105=1189.650,153.229,-54.766,-178.256,6.310,148.628
C07106=1189.645,153.478,-54.787,-178.254,6.310,148.628
C07107=1189.640,153.727,-54.808,-178.251,6.312,148.627
C07108=1189.635,153.976,-54.830,-178.248,6.314,148.627
C07109=1189.630,154.225,-54.850,-178.246,6.316,148.627
C07110=1189.626,154.474,-54.872,-178.242,6.317,148.626
C07111=1189.621,154.723,-54.893,-178.240,6.319,148.626
C07112=1189.616,154.972,-54.915,-178.238,6.320,148.625
C07113=1189.611,155.221,-54.936,-178.235,6.322,148.625
C07114=1189.607,155.470,-54.957,-178.232,6.324,148.625
C07115=1189.602,155.720,-54.978,-178.230,6.325,148.624
C07116=1189.597,155.968,-55.000,-178.227,6.327,148.624
C07117=1189.593,156.218,-55.021,-178.224,6.329,148.623
C07118=1189.588,156.467,-55.043,-178.222,6.329,148.623
C07119=1189.583,156.715,-55.065,-178.219,6.331,148.622
C07120=1189.578,156.964,-55.085,-178.216,6.333,148.622
C07121=1189.574,157.214,-55.107,-178.214,6.335,148.622
C07122=1189.569,157.463,-55.128,-178.211,6.337,148.621
C07123=1189.564,157.712,-55.150,-178.208,6.338,148.621
C07124=1189.560,157.961,-55.172,-178.206,6.340,148.621
C07125=1189.555,158.210,-55.193,-178.203,6.341,148.620
C07126=1189.550,158.479,-55.216,-178.200,6.342,148.620
C07127=1189.545,158.748,-55.240,-178.197,6.345,148.619
C07128=1189.540,159.017,-55.262,-178.194,6.347,148.619
C07129=1189.535,159.286,-55.287,-178.192,6.349,148.618
C07130=1189.530,159.535,-55.307,-178.188,6.350,148.618
C07131=1189.525,159.784,-55.329,-178.186,6.351,148.617
C07132=1189.521,160.033,-55.351,-178.184,6.353,148.617
C07133=1189.516,160.282,-55.372,-178.181,6.355,148.617
C07134=1189.511,160.531,-55.393,-178.178,6.356,148.616
C07135=1189.507,160.780,-55.415,-178.176,6.358,148.616
C07136=1189.502,161.029,-55.437,-178.173,6.360,148.616
C07137=1189.497,161.277,-55.459,-178.170,6.362,148.615
C07138=1189.493,161.527,-55.480,-178.168,6.363,148.615
C07139=1189.488,161.776,-55.502,-178.165,6.364,148.614
C07140=1189.484,162.025,-55.524,-178.162,6.366,148.614
C07141=1189.479,162.274,-55.545,-178.160,6.368,148.614
C07142=1189.474,162.522,-55.567,-178.157,6.369,148.613
C07143=1189.470,162.772,-55.589,-178.154,6.371,148.613
C07144=1189.464,163.021,-55.610,-178.152,6.373,148.612
C07145=1189.460,163.270,-55.632,-178.149,6.375,148.612
C07146=1189.455,163.519,-55.654,-178.146,6.377,148.612
C07147=1189.450,163.768,-55.676,-178.144,6.378,148.611
C07148=1189.446,164.017,-55.698,-178.141,6.379,148.611
C07149=1189.441,164.266,-55.719,-178.139,6.381,148.611
C07150=1189.436,164.515,-55.742,-178.136,6.383,148.610
C07151=1189.431,164.764,-55.764,-178.133,6.385,148.610
C07152=1189.427,165.013,-55.786,-178.131,6.386,148.609
C07153=1189.422,165.262,-55.807,-178.128,6.388,148.609
C07154=1189.418,165.511,-55.829,-178.125,6.390,148.608
C07155=1189.413,165.760,-55.851,-178.122,6.391,148.608
C07156=1189.408,166.009,-55.873,-178.120,6.393,148.608
C07157=1189.404,166.258,-55.895,-178.117,6.395,148.607
C07158=1189.399,166.507,-55.916,-178.115,6.396,148.607
C07159=1189.395,166.756,-55.939,-178.112,6.398,148.607
C07160=1189.390,167.005,-55.960,-178.109,6.400,148.606
C07161=1189.385,167.254,-55.983,-178.107,6.401,148.606
C07162=1189.380,167.503,-56.005,-178.104,6.403,148.605
C07163=1189.376,167.752,-56.027,-178.101,6.405,148.605
C07164=1189.371,168.001,-56.048,-178.099,6.407,148.605
C07165=1189.367,168.250,-56.070,-178.096,6.408,148.604
C07166=1189.362,168.499,-56.092,-178.093,6.410,148.604
C07167=1189.357,168.748,-56.115,-178.091,6.412,148.604
C07168=1189.352,168.996,-56.137,-178.088,6.414,148.603
C07169=1189.348,169.246,-56.159,-178.085,6.416,148.603
C07170=1189.343,169.494,-56.181,-178.083,6.417,148.603
C07171=1189.338,169.744,-56.203,-178.081,6.418,148.602
C07172=1189.333,169.993,-56.225,-178.078,6.420,148.602
C07173=1189.329,170.242,-56.247,-178.075,6.422,148.601
C07174=1189.324,170.490,-56.270,-178.073,6.424,148.601
C07175=1189.320,170.739,-56.292,-178.070,6.425,148.601
C07176=1189.315,170.988,-56.314,-178.067,6.427,148.600
C07177=1189.310,171.238,-56.336,-178.064,6.429,148.600
C07178=1189.306,171.487,-56.358,-178.061,6.430,148.599
C07179=1189.301,171.735,-56.381,-178.059,6.432,148.599
C07180=1189.296,171.985,-56.403,-178.056,6.434,148.599
C07181=1189.292,172.233,-56.425,-178.053,6.436,148.598
C07182=1189.287,172.483,-56.447,-178.051,6.438,148.598
C07183=1189.282,172.731,-56.470,-178.048,6.439,148.598
C07184=1189.278,172.980,-56.492,-178.045,6.441,148.597
C07185=1189.273,173.230,-56.514,-178.043,6.443,148.597
C07186=1189.268,173.478,-56.537,-178.040,6.445,148.596
C07187=1189.264,173.727,-56.559,-178.037,6.447,148.596
C07188=1189.259,173.976,-56.581,-178.035,6.448,148.596
C07189=1189.254,174.225,-56.604,-178.033,6.449,148.595
C07190=1189.250,174.474,-56.626,-178.030,6.451,148.595
C07191=1189.245,174.723,-56.648,-178.027,6.453,148.595
C07192=1189.240,174.972,-56.671,-178.025,6.455,148.594
C07193=1189.236,175.221,-56.693,-178.022,6.456,148.594
C07194=1189.231,175.470,-56.716,-178.019,6.458,148.594
C07195=1189.227,175.719,-56.738,-178.017,6.460,148.593
C07196=1189.222,175.967,-56.760,-178.014,6.462,148.593
C07197=1189.217,176.217,-56.783,-178.011,6.464,148.592
C07198=1189.213,176.466,-56.805,-178.009,6.465,148.592
C07199=1189.207,176.714,-56.828,-178.006,6.467,148.592
C07200=1189.203,176.964,-56.850,-178.003,6.469,148.591
C07201=1189.199,177.213,-56.874,-178.000,6.471,148.591
C07202=1189.194,177.461,-56.895,-177.998,6.473,148.591
C07203=1189.190,177.710,-56.918,-177.995,6.474,148.590
C07204=1189.185,177.960,-56.941,-177.992,6.476,148.590
C07205=1189.180,178.208,-56.963,-177.990,6.478,148.590
C07206=1189.175,178.458,-56.986,-177.988,6.480,148.589
C07207=1189.171,178.706,-57.008,-177.985,6.482,148.589
C07208=1189.166,178.955,-57.032,-177.982,6.484,148.589
C07209=1189.162,179.204,-57.053,-177.980,6.485,148.588
C07210=1189.157,179.453,-57.077,-177.977,6.487,148.588
C07211=1189.153,179.702,-57.099,-177.974,6.489,148.588
C07212=1189.147,179.951,-57.122,-177.972,6.491,148.587
C07213=1189.143,180.199,-57.145,-177.969,6.493,148.587
C07214=1189.138,180.449,-57.167,-177.966,6.494,148.587
C07215=1189.134,180.698,-57.190,-177.964,6.496,148.586
C07216=1189.129,180.946,-57.213,-177.961,6.498,148.586
C07217=1189.124,181.196,-57.236,-177.958,6.500,148.586
C07218=1189.120,181.444,-57.258,-177.956,6.501,148.585
C07219=1189.115,181.693,-57.282,-177.953,6.503,148.585
C07220=1189.111,181.942,-57.304,-177.950,6.505,148.584
C07221=1189.106,182.191,-57.327,-177.948,6.507,148.584
C07222=1189.102,182.440,-57.350,-177.945,6.509,148.584
C07223=1189.097,182.689,-57.372,-177.942,6.510,148.583
C07224=1189.092,182.938,-57.395,-177.940,6.512,148.583
C07225=1189.088,183.187,-57.418,-177.937,6.514,148.583
C07226=1189.083,183.436,-57.441,-177.934,6.516,148.582
C07227=1189.079,183.684,-57.464,-177.932,6.518,148.582
C07228=1189.074,183.934,-57.487,-177.929,6.520,148.582
C07229=1189.069,184.182,-57.510,-177.927,6.522,148.581
C07230=1189.064,184.452,-57.534,-177.923,6.524,148.581
C07231=1189.059,184.721,-57.559,-177.920,6.526,148.581
C07232=1189.053,184.991,-57.584,-177.918,6.527,148.580
C07233=1189.049,185.261,-57.609,-177.914,6.530,148.580
C07234=1189.044,185.510,-57.632,-177.912,6.532,148.580
C07235=1189.039,185.759,-57.655,-177.909,6.534,148.579
C07236=1189.035,186.007,-57.678,-177.906,6.535,148.579
C07237=1189.031,186.257,-57.702,-177.904,6.538,148.579
C07238=1189.025,186.505,-57.725,-177.902,6.539,148.578
C07239=1189.022,186.754,-57.747,-177.899,6.541,148.578
C07240=1189.017,187.003,-57.771,-177.896,6.543,148.578
C07241=1189.012,187.252,-57.794,-177.894,6.545,148.577
C07242=1189.007,187.501,-57.817,-177.891,6.547,148.577
C07243=1189.003,187.749,-57.840,-177.888,6.548,148.577
C07244=1188.999,187.998,-57.864,-177.886,6.550,148.576
C07245=1188.993,188.247,-57.887,-177.883,6.552,148.576
C07246=1188.988,188.496,-57.909,-177.880,6.554,148.575
C07247=1188.984,188.745,-57.932,-177.878,6.555,148.575
C07248=1188.980,188.994,-57.956,-177.875,6.558,148.575
C07249=1188.975,189.243,-57.979,-177.873,6.559,148.575
C07250=1188.971,189.492,-58.003,-177.870,6.561,148.574
C07251=1188.966,189.741,-58.026,-177.867,6.563,148.574
C07252=1188.961,189.990,-58.049,-177.864,6.566,148.574
C07253=1188.957,190.238,-58.072,-177.861,6.567,148.573
C07254=1188.953,190.487,-58.096,-177.859,6.569,148.573
C07255=1188.947,190.736,-58.119,-177.856,6.571,148.573
C07256=1188.943,190.985,-58.142,-177.853,6.573,148.572
C07257=1188.938,191.234,-58.165,-177.851,6.575,148.572
C07258=1188.933,191.483,-58.189,-177.849,6.577,148.572
C07259=1188.929,191.732,-58.212,-177.846,6.579,148.571
C07260=1188.925,191.980,-58.235,-177.843,6.580,148.571
C07261=1188.920,192.229,-58.259,-177.841,6.582,148.571
C07262=1188.915,192.478,-58.282,-177.838,6.584,148.570
C07263=1188.911,192.727,-58.306,-177.835,6.586,148.570
C07264=1188.906,192.976,-58.329,-177.832,6.588,148.570
C07265=1188.901,193.225,-58.352,-177.829,6.590,148.569
C07266=1188.897,193.474,-58.376,-177.827,6.592,148.569
C07267=1188.892,193.723,-58.400,-177.825,6.594,148.569
C07268=1188.888,193.972,-58.423,-177.822,6.596,148.568
C07269=1188.883,194.221,-58.446,-177.819,6.598,148.568
C07270=1188.878,194.469,-58.471,-177.817,6.600,148.568
C07271=1188.874,194.718,-58.494,-177.814,6.601,148.567
C07272=1188.869,194.967,-58.517,-177.811,6.603,148.567
C07273=1188.865,195.216,-58.541,-177.809,6.605,148.567
C07274=1188.860,195.465,-58.565,-177.806,6.608,148.567
C07275=1188.855,195.714,-58.588,-177.803,6.610,148.566
C07276=1188.851,195.963,-58.611,-177.801,6.611,148.566
C07277=1188.846,196.211,-58.635,-177.798,6.613,148.566
C07278=1188.841,196.460,-58.659,-177.795,6.615,148.565
C07279=1188.837,196.709,-58.683,-177.793,6.617,148.565
C07280=1188.832,196.958,-58.706,-177.790,6.619,148.565
C07281=1188.828,197.207,-58.730,-177.788,6.621,148.564
C07282=1188.823,197.455,-58.754,-177.785,6.623,148.564
C07283=1188.819,197.704,-58.777,-177.782,6.625,148.564
C07284=1188.814,197.952,-58.801,-177.779,6.627,148.563
C07285=1188.810,198.201,-58.824,-177.776,6.629,148.563
C07286=1188.805,198.450,-58.848,-177.774,6.631,148.563
C07287=1188.800,198.699,-58.872,-177.772,6.633,148.563
C07288=1188.796,198.948,-58.895,-177.769,6.635,148.562
C07289=1188.791,199.196,-58.919,-177.766,6.636,148.562
C07290=1188.787,199.446,-58.943,-177.763,6.639,148.562
C07291=1188.782,199.695,-58.968,-177.760,6.641,148.561
C07292=1188.777,199.944,-58.991,-177.758,6.643,148.561
C07293=1188.773,200.192,-59.015,-177.756,6.645,148.561
C07294=1188.768,200.441,-59.039,-177.753,6.647,148.560
C07295=1188.764,200.690,-59.063,-177.750,6.648,148.560
C07296=1188.759,200.939,-59.086,-177.748,6.650,148.560
C07297=1188.755,201.187,-59.110,-177.745,6.653,148.560
C07298=1188.750,201.436,-59.135,-177.742,6.655,148.559
C07299=1188.746,201.686,-59.158,-177.740,6.657,148.559
C07300=1188.741,201.934,-59.182,-177.737,6.659,148.559
C07301=1188.736,202.183,-59.206,-177.734,6.660,148.558
C07302=1188.732,202.431,-59.230,-177.732,6.662,148.558
C07303=1188.727,202.680,-59.255,-177.729,6.664,148.558
C07304=1188.722,202.929,-59.278,-177.726,6.667,148.557
C07305=1188.718,203.178,-59.302,-177.723,6.669,148.557
C07306=1188.714,203.427,-59.326,-177.721,6.671,148.557
C07307=1188.709,203.676,-59.350,-177.719,6.673,148.557
C07308=1188.704,203.924,-59.374,-177.716,6.674,148.556
C07309=1188.700,204.173,-59.399,-177.713,6.676,148.556
C07310=1188.695,204.422,-59.422,-177.710,6.679,148.556
C07311=1188.691,204.671,-59.446,-177.707,6.681,148.555
C07312=1188.686,204.920,-59.471,-177.705,6.683,148.555
C07313=1188.682,205.168,-59.495,-177.703,6.685,148.555
C07314=1188.677,205.417,-59.518,-177.700,6.686,148.554
C07315=1188.672,205.666,-59.543,-177.697,6.688,148.554
C07316=1188.668,205.915,-59.568,-177.694,6.691,148.554
C07317=1188.664,206.163,-59.592,-177.692,6.693,148.554
C07318=1188.659,206.412,-59.616,-177.689,6.695,148.553
C07319=1188.654,206.661,-59.640,-177.687,6.697,148.553
C07320=1188.650,206.910,-59.664,-177.684,6.698,148.553
C07321=1188.645,207.159,-59.689,-177.681,6.701,148.553
